	4: //Read back calibration file
		powermoduleCalib.b_StartCalibration := FALSE;
		pulseTimer(IN := NOT JsonFileToStruct(
			bExecute := pulseTimer.Q,
			sJsonPathName := 'C:\PLCUtility\CalDat_Powerstack.json',
			sStructName := 'ST_Powerstack_Calibration',
			pStruct := ADR(st_calibration.Powerstack),
			nStruct := SIZEOF(st_calibration.Powerstack),
			WriteMode := FALSE,
			sMessage => Message,
			Error => bError,
			Busy => bBusy
			));
		IF NOT pulseTimer.IN THEN
			SFCstep := 99;
		END_IF
		
	99: //clear all states for next round
		Error := bError; 
		sMessage := Message;
		pulseTimer.IN := FALSE;
		fbExecuteCalibrationFit(START := FALSE);
		DelayTimer.IN := FALSE;
		fbExecuteCalibrationFit.START := FALSE;
		PowerstackCalibration := TRUE;
		SFCstep := 0;
END_CASE
END_METHOD

METHOD Reset : BOOL
Reset := GenGridControl.Reset();
END_METHOD

METHOD SetPQLimits

VAR_INPUT
	r_BatPchargeLim			: REAL;
	r_BatPdischargeLim		: REAL;
	b_BatteryFull			: BOOL;
	b_BatteryEmpty			: BOOL;
	r_ACLinevoltage			: REAL;
	r_PchargeLimHard		: REAL;
	r_PchargeLimSoft		: REAL;
	r_PDischargeLimHard		: REAL;
	r_PDischargeLimSoft		: REAL;
	r_SmaxHard				: REAL;	//kVA
	r_AmaxHard				: REAL; //current
	r_AmaxSoft				: REAL; //current
END_VAR

VAR_OUTPUT
	r_Pmin				: REAL;
	r_PMax				: REAL;
	r_AMax				: REAL;
END_VAR

VAR_INST
	fb_rampPcharge						: FB_ramp := (b_enable := TRUE, r_ramprate := 25);
	fb_rampPdischarge					: FB_ramp := (b_enable := TRUE, r_ramprate := 25);
	fb_rampCurrentLimit					: FB_ramp := (b_enable := TRUE, r_ramprate := 100);
	
	r_BatChargeCorrectionFactor			: REAL := 0.98; // compensates inverter losses and BMS measurement errors
	r_BatDischargeCorrectionFactor		: REAL := 0.99;
	r_Smax								: REAL;
	r_PDischargeLimitUser				: REAL; //Discharging
	r_PChargeLimitUser					: REAL; //Charging
	r_AmaxLimitUser						: REAL;
	r_PmaxbySmax						: REAL;
	r_BatChargePowerLimitCalc			: REAL;
	r_BatDischargePowerLimitCalc		: REAL;
END_VAR
//user soft limit
fb_rampPcharge(IN := LIMIT(0 ,r_PchargeLimSoft, r_PchargeLimHard));
fb_rampPdischarge(IN := LIMIT(0,r_PDischargeLimSoft, r_PDischargeLimHard));

//current limit
r_AmaxLimitUser := MAX(0, KwToCurrent(r_SmaxHard,r_acLineVoltage), r_AmaxHard);
fb_rampCurrentLimit(IN := LIMIT(0,r_Amaxsoft, r_AmaxLimitUser), Q=> r_AMax);

r_Smax:= CurrentToKw(r_Amax, r_AClinevoltage);
r_PmaxbySmax := r_SMax; //SQRT(MAX(EXPT(r_Smax,2) - EXPT(r_ReaPower, 2),0));

//Set system Variable
r_Pmin := -MIN(ABS(r_BatPchargeLim / r_BatChargeCorrectionFactor), fb_rampPcharge.Q, r_PmaxbySmax);
r_Pmax := MIN(ABS(r_BatPdischargeLim * r_BatDischargeCorrectionFactor),  fb_rampPdischarge.Q, r_PmaxbySmax);

IF b_BatteryFull THEN
	r_Pmin := 0;
ELSIF b_BatteryEmpty THEN
	r_Pmax := 0; //overwrite value from input to 0.
END_IF
END_METHOD

METHOD shutdown : BOOL
VAR_INPUT
END_VAR

VAR_INST
	started : BOOL;
	ton_RetryDelay : TON := (PT := T#2s);
END_VAR
ton_RetryDelay(IN := TRUE);

IF storeSettings(ton_RetryDelay.Q, FALSE) THEN
	shutdown := TRUE;
	ton_RetryDelay(IN := FALSE);
END_IF
END_METHOD

METHOD StoreSettings : BOOL
VAR_INPUT
	execute : BOOL;
	writeMode: BOOL;
END_VAR

VAR_INST
	rTrigExecute	: R_TRIG;
	b_next : BOOL;
	sfcStep	: BYTE;
	tDelaySFCstep		: TON :=(PT := T#10MS);
END_VAR
rTrigExecute(CLK := execute);
IF rTrigExecute.Q THEN
	SFCstep := 1;
END_IF

CASE SFCstep OF
	1: b_next := JsonFileToStruct(
		bExecute := TRUE,
		sJsonPathName := 'C:\PLCUtility\MachineSettings.json',
		sStructName := 'ST_System_MachineParams',
		pStruct := ADR(settings.MachineParams),
		nStruct := SIZEOF(settings.MachineParams),
		WriteMode := writeMode,
		sMessage => sMessage
		);
	2: b_next := JsonFileToStruct(
		bExecute := TRUE,
		sJsonPathName := 'C:\PLCUtility\MachineConfig.json',
		sStructName := 'ST_System_Config',
		pStruct := ADR(settings.Configuration),
		nStruct := SIZEOF(settings.Configuration),
		WriteMode := writeMode,
		sMessage => sMessage
		);
	 3: b_next := JsonFileToStruct(
		bExecute := TRUE,
		sJsonPathName := 'C:\PLCUtility\GridSettings.json',
		sStructName := 'ST_System_GridCodeParams',
		pStruct := ADR(settings.GridParams),
		nStruct := SIZEOF(settings.GridParams),
		WriteMode := writeMode,
		sMessage => sMessage
		);
	 4: b_next := JsonFileToStruct(
		bExecute := TRUE,
		sJsonPathName := 'C:\PLCUtility\MachineProperties.json',
		sStructName := 'ST_System_Properties',
		pStruct := ADR(settings.Properties),
		nStruct := SIZEOF(settings.Properties),
		WriteMode := writeMode,
		sMessage => sMessage
		);
	5: b_next := JsonFileToStruct(
		bExecute := TRUE,
		sJsonPathName := 'C:\PLCUtility\CalDat_Powerstack.json',
		sStructName := 'ST_System_Calibration',
		pStruct := ADR(settings.Calibration),
		nStruct := SIZEOF(settings.Calibration),
		WriteMode := FALSE,
		sMessage => sMessage
		);
	ELSE
		SFCstep := 0;
		rTrigExecute(CLK := FALSE);
		StoreSettings := TRUE;	
END_CASE


IF b_next THEN 
	tDelaySFCstep(IN := TRUE);
 	IF tDelaySFCstep.q THEN 
	SFCstep := SFCstep + 1;
		tDelaySFCstep(IN := FALSE);
	END_IF 
END_IF
END_METHOD

METHOD UpdateSystemTime : BOOL
VAR_INST
	SetTime :	NT_SetLocalTime();
	rtrig_AutoUpdate	:	r_Trig;
	ftrig_UpdateDone	:	f_Trig;
	systime				:	Timestruct;

	SystemTimeStamp		:	DINT;
	GPSTimeStamp		:	DINT;
	TON_GpsUpdateReq	:	TON := (PT := T#5M); 
	
	NewTimeString		:	STRING;
	NewTimeStruct		:	Timestruct;

	
	UpdateRequired		:	BOOL;
END_VAR

monitor.system.DT_SystemTime := GVL.dt_SystemDateTime;

//first fix datetime format from teltonika.
IF st_params.SystemTime.AutoSyncToGPS THEN 
	TON_GpsUpdateReq(in := ABS(DT_TO_DINT(monitor.router.GPS.DateTime) - DT_TO_DINT(gvl.dt_SystemDateTime)) > 30);
	IF ton_gpsUpdateReq.Q THEN
		NewTimeStruct := DT_TO_Systemtime(monitor.Router.GPS.DateTime);
		UpdateRequired	:=	TRUE;
	ELSE
		UpdateRequired	:=	FALSE;
	END_IF
ELSE
	IF st_params.SystemTime.ManualSync THEN
		st_params.SystemTime.ManualSync := FALSE;
		NewTimeStruct := DT_TO_SYSTEMTIME(st_params.SystemTime.ManSyncValue);
		UpdateRequired	:=	TRUE;
	END_IF
END_IF
	
SetTime(	TimeSTR := NewTimeStruct, //convert to Systemtime struct and write to plc
	start	:= UpdateRequired,
	TMOUT	:= T#1S);

			
ftrig_UpdateDone(clk := SetTime.BUSY);

IF ftrig_UpdateDone.Q THEN
	UpdateRequired := FALSE;
	monitor.system.events.b_TimeUpdateFailed := FALSE;
	IF SetTime.ERR THEN
		monitor.system.events.b_TimeUpdateFailed := TRUE;
	END_IF
END_IF
END_METHOD

END_FUNCTION_BLOCK

// ---- POUs/System/PowerControl/FB_PowerControl.TcPOU
FUNCTION_BLOCK FB_PowerControl
VAR_IN_OUT CONSTANT						
	powerstack							: ST_Powerstack_get;
	powermonitor						: ST_powermonitor_get;
	st_params							: ST_Powercontrol_Params;
END_VAR

VAR_INPUT
	r_Soc								: REAL;
	r_SocMin							: REAL;
	r_SocMax							: REAL;
	b_calibrationRun					: BOOL;
	
	
	//inverter data	
	Target								: ST_PowerControl_Target; //input from gengrid controller
	
	r_Pset								: REAL;
	r_Qset								: REAL;
	r_PFset								: REAL;
	b_PFsetEnable						: BOOL;	
	r_Frequency							: REAL;
	r_FreqDroop							: REAL;
	r_Voltage							: REAL;
	r_VoltDroop							: REAL;
	b_GensetLoadshareControl			: BOOL;
	r_GenfixPowerTarget					: REAL;
	r_GenRatedPower						: REAL;
	b_GenStarted						: BOOL;
END_VAR

VAR_OUTPUT
	r_ActivePowerRQInv			: REAL; // Positive discharging, negative charging
	r_ReactivePowerRQInv		: REAL; // Positive  Inductive, negative Capacitive
	r_ActivePowerRQGen			: REAL;
	r_ReactivePowerRQGen		: REAL;
	b_ExtSyncingActive			: BOOL;
	r_FrequencyRQ				: REAL;
	r_VoltageRQ					: REAL;
	r_FreqDroopRQ				: REAL;
	r_VoltDroopRQ				: REAL;
END_VAR
VAR_OUTPUT
	get							: ST_PowerControl_Get;
END_VAR
VAR	
	//General
	VoltageOK				: fbValueOutOfRange;
	ActiveOK				: fbValueOutOfRange;
	ReactiveOK				: fbValueOutOfRange;
	
	//Controlvars
	r_ManSyncPower			: REAL;
	b_Sync					: BOOL;
	r_ReactiveSetpoint		: REAL := 0;
	b_ReactivePIDLimitReached : BOOL;
	
	GensetPeakshaverEnable 	: BOOL;
	r_ActiveSetpoint		: REAL := 0;
	b_ActivePIDLimitReached : BOOL;
	e_ctrl					: e_CTRL_MODE;
	
	b_ReactiveLimit			: BOOL;
	b_ActiveLimit			: BOOL;
END_VAR

//get measured data from peakshaver target or bess netto output.
TargetSection();

//Determine Reactive power setpoint
r_ReactiveSetpoint := PFtoReactiveSetpoint(
	enable := b_PFsetEnable,
	forcezeroQ:= target.b_GenIsoPID,
	voltage := powerstack.r_ACVoltageD7,
	AcCurrentLimit := MAX(target.r_FeedInCurrentLimit, target.r_SupplyCurrentLimit),
	Sact:= get.r_Sact, 
	Qset:= r_Qset,
	PFset:= r_PFset);

//Use droop controller if inverter is in droop mode.
//IF powerstack.e_InverterMode <> eInverterModes.AFE AND powerstack.Netcontactor.b_NetConFb THEN
	DroopController(
		r_NomVolt	:= r_Voltage,
		r_NomFreq	:= r_Frequency,
		r_FreqDroop	:= r_FreqDroop,
		r_VoltDroop	:= r_VoltDroop,
		b_EnableSocDrooping		:= Target.b_EnableSocDrooping AND st_params.SocDroop.enable AND powerstack.b_StartedState,
		r_FreqRQ 		=> r_FrequencyRQ, 
		r_voltRQ 		=> r_VoltageRQ,
		r_FreqDroopRQ	=> r_FreqDroopRQ,
		r_VoltDroopRQ 	=> r_VoltDroopRQ
);
//for letting now powermodule.
b_ExtSyncingActive := target.Syncdata.b_Sync;

//Peakshave power PID controller
IF b_calibrationRun THEN
	Target.PIDmode := ePIDMode.None;
END_IF
PeakshaveController(VoltageOK.Q, ActiveOK.Q, ReactiveOK.Q, Target.PIDmode <> ePIDmode.None AND st_params.ActivePID.enable);

PIDcontrollers(
	b_Activate :=  powerstack.b_ControlEnabled AND powerstack.b_startedstate,
	b_QEnable := (Target.PIDmode = ePIDmode.Q OR Target.PIDmode = ePIDmode.Both) AND st_params.ReactivePID.enable,
	b_PEnable := (Target.PIDmode = ePIDmode.P OR Target.PIDmode = ePIDmode.Both) AND st_params.ActivePID.enable,
	);
	
GensetController(
	Enable := b_GensetLoadshareControl AND b_genstarted,
	GenRatedPower := r_GenRatedPower,
	PeakshaveMode := target.PeakshaveMode,
	ActiveControlEnable := b_activePIDLimitReached OR NOT powerstack.b_startedstate,
	ReactiveControlEnable := b_ReactivePIDLimitReached OR NOT powerstack.b_startedstate,
	Ptarget := -CurrentTokW(target.r_SupplyCurrentLimit, powermonitor.OutputField.ar_LineVoltage[0]),
	PAct := target.Measurements.r_ActivePower,
	PManSet := r_GenfixPowerTarget,
	Qtarget	:= -target.Measurements.r_ReactivePower,
	QactPID := r_ReactivePowerRQInv,
	Pset => r_ActivePowerRQGen,
	Qset => r_ReactivePowerRQGen);
	
//set throttling info	 
ThrottlingInfoSection();

METHOD PRIVATE DroopController : BOOL
VAR_INPUT
	r_NomVolt			: REAL;
	r_NomFreq			: REAL;
	r_FreqDroop			: REAL;
	r_VoltDroop			: REAL;
	b_EnableSocDrooping	: BOOL;
END_VAR

VAR_OUTPUT
	r_FreqRQ				: REAL;
	r_VoltRQ				: REAL;
	r_FreqDroopRQ			: REAL;
	r_VoltDroopRQ			: REAL;
END_VAR

VAR_INST
	b_master				: BOOL := TRUE;
	r_SoCMiddlepoint		: REAL;
	r_FreqZeroCharge		: REAL;
	r_FreqZeroDischarge		: REAL;
	r_SocStartFreqShiftDown : REAL;
	r_SocStartFreqShiftUp   : REAL;

	
	DroopRamp				: fb_ramp := (b_enable := TRUE);
	FreqRamp				: fb_ramp := (b_enable := TRUE);
	VoltRamp				: fb_ramp := (b_enable := TRUE);
	
	
	//freq shift PID
	r_DroopFreqMax			: REAL;
	FreqShiftPID			: fb_ctrl_pid_ext := (eMode := e_Ctrl_mode.eCTRL_MODE_ACTIVE);
	FreqShiftPID_params 	: ST_CTRL_PID_EXT_PARAMS := (
							tCtrlCycleTime := T#10MS,
							tTaskCycleTime := T#2MS);
	r_FreqShiftOut			: REAL;
	
	//Volt shift PID
	r_VoltMaxShiftDelta		: REAL := 40;		
	VoltShiftPID			: fb_ctrl_pid_ext := (eMode := e_Ctrl_mode.eCTRL_MODE_ACTIVE);
	VoltShiftPID_params 	: ST_CTRL_PID_EXT_PARAMS := (
							tCtrlCycleTime := T#10MS,
							tTaskCycleTime := T#2MS);
	r_VoltShiftOut			: REAL;
		
	
END_VAR
r_DroopFreqMax :=  MAX(0.01, powerstack.r_FrequencyDroop) / 100 * settings.GridParams.r_GridNominalFrequency;

r_FreqZeroCharge := r_NomFreq - r_DroopFreqMax;
r_FreqZeroDischarge := r_NomFreq + r_DroopFreqMax;
r_SocStartFreqShiftDown := MAX(r_SocMin, st_params.SocDroop.SocMinDroopStart);
r_SocStartFreqShiftUp   := MIN(r_SocMax, st_params.SocDroop.SocMaxDroopStart);

FreqRamp(r_rampRate := 0.5, SetToIN:= FreqRamp.Q < settings.GridParams.r_GridFrequencyMin);
VoltRamp(r_rampRate := 1, SetToIN := VoltRamp.Q < settings.GridParams.r_GridVoltageMin);
//Voltage set
VoltRamp.IN := LIMIT(settings.GridParams.r_GridVoltageMin, r_Nomvolt, settings.GridParams.r_GridVoltageMax);

//freq shift pid
	VoltShiftPID_params.fkp := st_params.FreqShiftPID.Kp;
	VoltShiftPID_params.tTd := TO_TIME(st_params.FreqShiftPID.Td);
	VoltShiftPID_params.tTn := TO_TIME(st_params.FreqShiftPID.Tn);
	VoltShiftPID_params.tTv := TO_TIME(st_params.FreqShiftPID.Tv);
	VoltShiftPID_params.fOuterWindow := st_params.FreqShiftPID.Outerwindow;
	VoltShiftPID_params.fInnerWindow := st_params.FreqShiftPID.Innerwindow;
	VoltShiftPID_params.fDeadBandOutput := st_params.FreqShiftPID.OutputDeadband;
	VoltShiftPID_params.fDeadBandInput := st_params.FreqShiftPID.InputDeadband;
	VoltShiftPID_params.fOutMaxLimit := r_VoltMaxShiftDelta;
	VoltShiftPID_params.fOutMinLimit := -r_VoltMaxShiftDelta;
	VoltShiftPID(
		fsetPointValue := 0,
		fActualValue := SEL(b_master, powerstack.r_ReactivePower, powerstack.r_ACVoltageD7 - r_NomVolt),
		(*fManSyncValue := powerstack.r_FrequencyD7 - r_NomFreq,
		bSync := FALSE,//powerstack.b_StartedState,*)
		stparams := VoltShiftPID_params);
		//activate simultaniously with freqshift pid.
	IF NOT VoltShiftPID.bError AND NOT target.Syncdata.b_Sync AND st_params.FreqShiftPID.enable AND powerstack.b_StartedState AND powerstack.b_InverterGridFormingMode THEN
		VoltShiftPID.eMode := e_Ctrl_Mode.eCTRL_MODE_ACTIVE;
		r_VoltShiftOut := VoltShiftPID.fOut;
	ELSE
		r_VoltShiftOut := 0;
		VoltShiftPID.eMode := e_Ctrl_Mode.eCTRL_MODE_RESET;
	END_IF
			
//linearly scale frequency down when within soc charge prio and soc min
IF r_soc < r_SocStartFreqShiftDown AND b_EnableSocDrooping THEN
	//Frequency set
	FreqRamp.IN := scale(
		r_in:=r_soc,
		 In_min:= r_SocMin,
		 In_max:= r_SocStartFreqShiftDown,
		 Out_min:= r_FreqZeroCharge,
		 Out_max:= r_NomFreq);
ELSIF r_Soc > r_SocStartFreqShiftUp AND b_EnableSocDrooping THEN
	//Frequency set
	FreqRamp.IN := scale(
		r_in:=r_soc,
		 In_min:= r_SocStartFreqShiftUp,
		 In_max:= r_Socmax,
		 Out_min:= r_NomFreq,
		 Out_max:= r_FreqZeroDischarge);
ELSE
	//Frequency set
	FreqRamp.IN := r_NomFreq;
END_IF

//r_SocFreqShift := FreqRamp.Q - r_NomFreq;

//freq shift pid
	FreqShiftPID_params.fkp := st_params.FreqShiftPID.Kp;
	FreqShiftPID_params.tTd := TO_TIME(st_params.FreqShiftPID.Td);
	FreqShiftPID_params.tTn := TO_TIME(st_params.FreqShiftPID.Tn);
	FreqShiftPID_params.tTv := TO_TIME(st_params.FreqShiftPID.Tv);
	FreqShiftPID_params.fOuterWindow := st_params.FreqShiftPID.Outerwindow;
	FreqShiftPID_params.fInnerWindow := st_params.FreqShiftPID.Innerwindow;
	FreqShiftPID_params.fDeadBandOutput := st_params.FreqShiftPID.OutputDeadband;
	FreqShiftPID_params.fDeadBandInput := st_params.FreqShiftPID.InputDeadband;
	FreqShiftPID_params.fOutMaxLimit := r_DroopFreqMax;
	FreqShiftPID_params.fOutMinLimit := -r_DroopFreqMax;
	FreqShiftPID(
		fsetPointValue := 0,
		fActualValue := powerstack.r_FrequencyD7 - r_NomFreq,
		(*fManSyncValue := powerstack.r_FrequencyD7 - r_NomFreq,
		bSync := FALSE,//powerstack.b_StartedState,*)
		stparams := FreqShiftPID_params);
			
IF NOT FreqShiftPID.bError AND st_params.FreqShiftPID.enable AND powerstack.b_StartedState AND powerstack.e_InverterMode = eInvertermodes.Microgrid THEN
	FreqShiftPID.eMode := e_Ctrl_Mode.eCTRL_MODE_ACTIVE;
	r_FreqShiftOut := FreqShiftPID.fOut;
ELSE
	r_FreqShiftOut := 0;
	FreqShiftPID.eMode := e_Ctrl_Mode.eCTRL_MODE_RESET;
END_IF

r_FreqRQ := LIMIT(r_FreqZerocharge, FreqRamp.Q + r_FreqShiftOut, r_FreqZerodisCharge);
r_VoltRQ := VoltRamp.Q + r_VoltshiftOut;

//overwrite if sync is called
DroopRamp(r_Ramprate := 0.5);
IF target.Syncdata.b_Sync THEN
	DroopRamp.IN :=0.5;
	r_FreqDroopRQ:= DroopRamp.Q;
	r_VoltDroopRQ:= DroopRamp.Q;
	r_freqRQ := target.Syncdata.r_freqSet;
	r_voltRQ := target.Syncdata.r_VoltSet;
ELSE
	DroopRamp.IN := r_FreqDroop;
	r_FreqDroopRQ := MAX(Target.r_droopMinimum,r_FreqDroop);
	r_VoltDroopRQ := MAX(Target.r_droopMinimum, r_VoltDroop);
END_IF
END_METHOD

METHOD EMstop : BOOL
VAR_INPUT
END_VAR
e_ctrl := e_CTRL_MODE.eCTRL_MODE_RESET;
r_ActivePowerRQInv := 0;
r_ReactivePowerRQInv := 0;
END_METHOD

METHOD GensetController : BOOL
VAR_INPUT
	Enable					: BOOL;
	GenRatedPower			: REAL; //kVA
	PeakshaveMode			: BOOL;
	ActiveControlEnable		: BOOL;
	ReactiveControlEnable 	: BOOL;
	PTarget					: REAL;
	PAct					: REAL;
	PManSet					: REAL;
	QTarget					: REAL;
	QActPID					: REAL;
END_VAR

VAR_INST
	//Active powercontrol
	PStepSize 				: REAL := 0.001; //kW
	PDelta					: REAL;
	Pcum					: REAL;
	PlimitReached			: BOOL;
	
	//Reactive powercontrol
	QStepSize 				: REAL := 0.001; //kvar
	QDelta					: REAL;
	Qcum					: REAL;
	

	PFmin					: REAL := 0.8;
	QLimit					: REAL;
	
	GenLimit				: REAL := 90; //%
END_VAR

VAR_OUTPUT
	Pset			: REAL; //in %
	Qset			: REAL; //in %
END_VAR
IF enable THEN
	
	IF ActiveControlEnable AND PeakshaveMode THEN
		PDelta := PTarget - PAct;
		Pcum := LIMIT(0, Pcum + LIMIT(-1, PDelta, 1)* PStepSize, GenLimit);
	ELSE
		Pcum := LIMIT(0, PManSet, ABS(powerstack.r_Pmin));
	END_IF
	
	 
	Qlimit := ABS(Pcum)* ACOS(PFmin);
	
	IF ReactiveControlEnable AND PeakshaveMode THEN
		QDelta := QTarget - QActPID;
		Qcum := LIMIT(-Qlimit, Qcum + QDelta* QStepSize, Qlimit);
	ELSE
		Qcum := 0;
	END_IF
ELSE
	Pcum:= 0;
	Qcum:= 0;
END_IF

Pset := LIMIT(0, Pcum / MAX(1, GenRatedPower) * 100, GenLimit);// percentage limit to 90% of gen power
Qset :=LIMIT(0, Qcum / MAX(1, GenRatedPower) * 100, GenLimit);
END_METHOD

METHOD GetDiagnostics : BOOL
VAR_IN_OUT
	AddError		: ARRAY [*] OF FB_AddErrorST;
	a_ActiveEvents	: ARRAY [*] OF ST_ErrorStruct;
	w_Index			: WORD;
END_VAR
(*Reactive PID error*) 	AddError[w_Index](
		b_ErrorTrig			:= Get.Events.b_ReactivePIDError,
		out_ST_Error			:= a_ActiveEvents[w_Index],
		w_ErrorID				:= 1,
		e_ObjectID				:= eObject_ID.PowerController,
		s_Message				:= 'Reactive PID controller fault.',
		e_sev					:= eseverity.Warning
		);
	w_Index := w_Index +1;
	
(*Active PID error*) 	AddError[w_Index](
		b_ErrorTrig			:= Get.Events.b_ActivePIDError,
		out_ST_Error			:= a_ActiveEvents[w_Index],
		w_ErrorID				:= 2,
		e_ObjectID				:= eObject_ID.PowerController,
		s_Message				:= 'Active PID controller fault.',
		e_sev					:= eseverity.Warning
		);
	w_Index := w_Index +1;
	
(*FreqShift PID error*) 	AddError[w_Index](
		b_ErrorTrig				:= Get.Events.b_ActivePIDError,
		out_ST_Error			:= a_ActiveEvents[w_Index],
		w_ErrorID				:= 3,
		e_ObjectID				:= eObject_ID.PowerController,
		s_Message				:= 'Frequency Shift PID controller fault.',
		e_sev					:= eseverity.Warning
		);
	w_Index := w_Index +1;
END_METHOD

METHOD PRIVATE PeakshaveController : BOOL
VAR_INPUT
	Voltage_OK		: BOOL;
	P_OK			: BOOL;
	Q_OK			: BOOL;
	Enable			: BOOL;
END_VAR

VAR_INST
	FeedLimitCorrection : REAL;
	SupplyLimitCorrection : REAL;
	
	ton_ResetZeroPower : TON := (PT := T#5S);
	r_AppPowerLimIntoSystem		: REAL;
	r_AppPowerLimOutOfSystem	: REAL;
	r_ActivePowerLimIntoSystem	: REAL;
	r_ActivePowerLimOutOfSystem	: REAL;	
	r_PowerDemand				: REAL;
	PIDOK						: BOOL;
	
	r_rampRate					: REAL;
	fbPlimIntoSysRamp			: FB_RAMP := (b_enable := TRUE, r_rampRate := 5); //kw per second)
	fbPlimOutOfSysRamp			: FB_RAMP := (b_enable := TRUE, r_rampRate := 5); //kw per second)
	
END_VAR
//Set slow ramp for genset
r_rampRate:= LIMIT(1, target.r_PIDRampRate, 100);
fbPlimIntoSysRamp(SetZero := NOT (powerstack.b_ControlEnabled AND PIDOK),  r_ramprate := r_rampRate, Q => r_ActivePowerLimIntoSystem,);
fbPlimOutOfSysRamp(SetZero := NOT (powerstack.b_ControlEnabled AND PIDOK), r_ramprate :=  r_rampRate, Q => r_ActivePowerLimOutOfSystem);
ton_ResetZeroPower();
ton_ResetZeroPower.IN := FALSE;

PIDOK := VoltageOK.Q AND ActiveOK.Q AND ReactiveOK.Q AND Enable;
VoltagePeakshavePID(enable:= PIDOK,
	PIDParams := st_params.VoltagePeakshavePID, 
	FeedinLimitCorrection => FeedLimitCorrection, 
	SupplyLimitCorrection => SupplyLimitCorrection);

//power controller sectio
IF PIDOK THEN
	b_Sync := FALSE;
	
	//get active power limits based on the current values.
	r_AppPowerLimIntoSystem := CurrentTokW(LIMIT(0, Target.r_SupplyCurrentLimit - SupplyLimitCorrection, Target.r_SupplyCurrentLimit), get.r_PhaseVoltageAct * 1.73);
	r_AppPowerLimOutOfSystem := CurrentTokW(LIMIT(0, Target.r_FeedInCurrentLimit + FeedLimitCorrection, Target.r_FeedInCurrentLimit), get.r_PhaseVoltageAct * 1.73);
	
	IF target.b_GenIsoPID THEN
		fbPlimIntoSysRamp.IN := r_AppPowerLimIntoSystem;
		fbPlimOutOfSysRamp.IN := r_AppPowerLimOutOfSystem;
	ELSE
		fbPlimIntoSysRamp.IN:= SQRT(ABS(EXPT(r_AppPowerLimIntoSystem,2) - EXPT(get.r_Qact,2))) * SEL(r_AppPowerLimIntoSystem < 0, 1, -1);
		fbPlimOutOfSysRamp.IN:= SQRT(ABS(EXPT(r_AppPowerLimOutOfSystem,2) - EXPT(get.r_Qact,2))) * SEL(r_AppPowerLimOutOfSystem < 0, 1, -1);
	END_IF
	
	r_PowerDemand	:= get.r_Pact - powerstack.r_ActivePower + Target.r_PowerTarget;
	r_activeSetpoint 	:= LIMIT(-r_ActivePowerLimIntoSystem, r_powerDemand, r_ActivePowerLimOutOfsystem);
	
ELSE //If measurements not OK or peakshave target disabled, set manually values.
	//RESET some values
	r_activeSetpoint := r_Pset;
END_IF
END_METHOD

METHOD PRIVATE PFToReactiveSetpoint : REAL
VAR_INPUT
	enable 			: BOOL;
	ForceZeroQ		: BOOL;
	voltage			: REAL;
	Sact			: REAL;
	Qset			: REAL;
	AcCurrentLimit	: REAL;
	PFset			: REAL;
END_VAR

VAR_INST
	PFlimited 	: REAL;
	ReactiveSetpoint	: REAL;
	ApparentPowerLimit: REAL;
END_VAR
ApparentPowerLimit := CurrentToKw(AcCurrentLimit, voltage);

IF enable THEN
	PFlimited := LIMIT(-1, PFset, 1);
	ReactiveSetpoint := Sact * SQRT(1-EXPT(PFset,2))* SEL(PFset < 0, 1, -1);
ELSE
	ReactiveSetpoint := Qset;
END_IF

IF forcezeroQ THEN
	ReactiveSetpoint := 0;
END_IF

PFToReactiveSetpoint := LIMIT(-ApparentPowerLimit, ReactiveSetpoint, ApparentPowerLimit);
END_METHOD

METHOD PRIVATE PIDcontrollers : BOOL

VAR_INPUT
	b_Activate							: BOOL;
	b_QEnable							: BOOL;
	b_PEnable							: BOOL;
END_VAR

VAR_INST
	tnActive					: UINT;
	tnReactive					: UINT;
	
	//triggers
	tonPIDStartDelay		: TON := (PT := T#2S);
	tofPIDSyncHoldDelay		: Tof ;
	r_TriggerReactivePIDMode: R_Trig;
	r_TriggerActivePIDMode	: R_Trig;
	r_TriggerPIDHmiReset	: R_Trig;
	f_TriggerPIDHmiActivate	: F_TRIG;
	
	//Reactive PID
	TranstionReactivePowerRamp			: fb_ramp;	
	fb_PIDReactiveCurrent				: FB_CTRL_PID_EXT;
	st_Params_Reactive					: ST_CTRL_PID_EXT_PARAMS;
	
	
	//Active PID
	TranstionActivePowerRamp			: fb_ramp;
	TransitionSync						: BOOL;	
	fb_PIDActiveCurrent					: FB_CTRL_PID_EXT;
	st_Params_Active					: ST_CTRL_PID_EXT_PARAMS;
	b_DinFbPath							: BOOL; 
	b_ActiveLimitReached				: BOOL;
END_VAR
//set PID RESET/ACTIVE TRIGGER when inverter is running
tonPIDStartDelay(IN:= b_Activate);
tofPIDSyncHoldDelay(IN := target.Syncdata.b_Sync, PT := TO_TIME(st_params.TransitionTime));
r_TriggerReactivePIDMode(CLK:= tonPIDStartDelay.Q AND b_QEnable AND NOT tofPIDSyncHoldDelay.Q);
r_TriggerActivePIDMode(CLK:= tonPIDStartDelay.Q AND b_PEnable AND NOT tofPIDSyncHoldDelay.Q);

IF target.b_GenIsoPID THEN
	tnActive := MAX(100, st_params.ActivePID.Tn * 5);
	tnReactive := MAX(100, st_params.ReactivePID.Tn * 5);
ELSE
	tnActive := st_params.ActivePID.Tn;
	tnReactive := st_params.ReactivePID.Tn;
END_IF


IF r_TriggerReactivePIDMode.CLK THEN
	fb_PIDReactiveCurrent.eMode := e_CTRL_MODE.eCTRL_MODE_ACTIVE;
END_IF

IF r_TriggerActivePIDMode.CLK THEN
	fb_PIDActiveCurrent.eMode := e_CTRL_MODE.eCTRL_MODE_ACTIVE;
END_IF

//RESETS
IF NOT b_PEnable OR NOT b_Activate OR e_ctrl = e_CTRL_MODE.eCTRL_MODE_Reset THEN
	fb_PIDActiveCurrent.eMode := e_CTRL_MODE.eCTRL_MODE_Reset;
END_IF
IF NOT b_QEnable OR NOT b_Activate OR e_ctrl = e_CTRL_MODE.eCTRL_MODE_Reset THEN
	fb_PIDReactiveCurrent.eMode := e_CTRL_MODE.eCTRL_MODE_Reset;
END_IF

//r_TriggerPIDHmiReset(CLK := st_params.PIDreset);
//IF r_triggerPIDHmiReset.Q THEN
//	fb_PIDActiveCurrent.eMode := e_CTRL_MODE.eCTRL_MODE_Reset;
//	fb_PIDReactiveCurrent.eMode := e_CTRL_MODE.eCTRL_MODE_Reset;
//END_IF

//f_TriggerPIDHmiActivate(CLK:= st_params.PIDreset);
//IF f_triggerPIDHmiActivate.Q THEN
//	fb_PIDActiveCurrent.eMode := e_CTRL_MODE.eCTRL_MODE_Active;
//	fb_PIDReactiveCurrent.eMode := e_CTRL_MODE.eCTRL_MODE_Active;
//END_IF

//fb_QlimitMA(IN := LIMIT(0, powerstack.r_Qmax - ABS(powerstack.r_ReactivePower), powerstack.r_Qmax));

	st_Params_reactive.tCtrlCycleTime 		:= T#1MS;
		st_Params_reactive.tTaskCycleTime 	:= T#1MS;
		st_Params_reactive.fKp				:= st_params.ReactivePID.Kp /100;
		st_Params_reactive.tTn				:= TO_TIME(tnReactive);
		st_Params_reactive.tTv				:= TO_TIME(st_params.ReactivePID.Tv);
		st_Params_reactive.tTd				:= TO_TIME(st_params.ReactivePID.Td);
		st_Params_reactive.fOutMaxLimit		:= powerstack.r_RatedPower;
		st_Params_reactive.fOutMinLimit		:= -powerstack.r_RatedPower;
		st_Params_reactive.fDeadBandInput	:=  st_params.ReactivePID.InputDeadband;
		st_Params_reactive.fDeadBandOutput	:=  st_params.ReactivePID.OutputDeadband; //
		st_Params_reactive.finnerwindow		:=  st_params.ReactivePID.Innerwindow; //
		st_Params_reactive.fOuterWindow		:=  st_params.ReactivePID.Outerwindow;
	
	
	fb_PIDReactiveCurrent(
		fSetpointValue 	:=r_ReactiveSetpoint,
		bError			=> get.events.b_ReactivePIDError,
		fActualValue	:= target.Measurements.r_ReactivePower,
		stParams		:=st_Params_reactive);
	
	b_ReactivePIDLimitReached := fb_PIDReactiveCurrent.bMaxLimitReached OR fb_PIDReactiveCurrent.bMinLimitReached;

		//when active PID is started, the sync value must be hold for a while. 
TranstionReactivePowerRamp(IN := powerstack.r_ReactivePower, b_enable:= TRUE, r_ramprate := st_params.TransitionRamp);
fb_PIDReactiveCurrent.fManSyncValue := TranstionReactivePowerRamp.Q;

IF fb_PIDReactiveCurrent.eMode = e_CTRL_MODE.eCTRL_MODE_ACTIVE AND NOT fb_PIDReactiveCurrent.bError THEN
	fb_PIDReactiveCurrent.bSync := TRUE;
	r_ReactivePowerRQInv := fb_PIDReactiveCurrent.fOut; 
ELSIF tofPIDSyncHoldDelay.Q THEN
	fb_PIDReactiveCurrent.bSync := FALSE;
	r_ReactivePowerRQInv := TranstionReactivePowerRamp.Q;
ELSE	
	fb_PIDReactiveCurrent.bSync := FALSE;
	r_ReactivePowerRQInv := r_ReactiveSetpoint;
END_IF


	//ACTIVE POWER PID
	st_Params_Active.tCtrlCycleTime 		:= T#1MS;
		st_Params_Active.tTaskCycleTime 	:= T#1MS;
		st_Params_Active.fKp				:= st_params.ActivePID.Kp / 100;
		st_Params_Active.tTn				:= TO_TIME(tnActive);
		st_Params_Active.tTv				:= TO_TIME(st_params.ActivePID.Tv);
		st_Params_Active.tTd				:= TO_TIME(st_params.ActivePID.Td);
		st_Params_Active.fOutMaxLimit		:= powerstack.r_Pmax;
		st_Params_Active.fOutMinLimit		:= powerstack.r_Pmin;
		st_params_Active.fDeadBandInput		:= st_params.ActivePID.InputDeadband;
		st_Params_Active.fDeadBandOutput	:= st_params.ActivePID.OutputDeadband; //kW
		st_Params_Active.bDInTheFeedbackPath := b_DinFbPath;
		st_params_ACtive.bPInTheFeedbackPath := FALSE;
		st_Params_Active.finnerwindow		:=  st_params.ActivePID.innerwindow;
		st_Params_Active.fOuterWindow		:=  st_params.ActivePID.Outerwindow;
			

	//Active Power PID
	fb_PIDActiveCurrent(
		 fSetpointValue := r_ActiveSetpoint,
		 fActualValue	:=	target.Measurements.r_ActivePower,
		 fManSyncValue := r_ManSyncPower,
		 bError			=> get.events.b_ActivePIDError,
		 stParams		:=st_Params_Active);

	b_ActivePIDLimitReached := fb_PIDactiveCurrent.bMaxLimitReached OR fb_PIDactiveCurrent.bMinLimitReached;
//when active PID is started, the sync value must be hold for a while. 
TranstionActivePowerRamp(IN := powerstack.r_ActivePower, b_enable:= TRUE, r_ramprate := st_params.TransitionRamp);
r_ManSyncPower := TranstionActivePowerRamp.Q;

IF fb_PIDActiveCurrent.eMode = e_CTRL_MODE.eCTRL_MODE_ACTIVE AND NOT fb_PIDActiveCurrent.bError THEN
	IF transitionsync THEN
		fb_PIDActiveCurrent.bSync := TRUE;
		transitionsync:= FALSE;
	ELSE
		fb_PIDActiveCurrent.bSync := b_sync;
	END_IF
	r_ActivePowerRQInv := fb_PIDActiveCurrent.fOut; 
ELSIF tofPIDSyncHoldDelay.Q THEN
	TransitionSync := TRUE;
	fb_PIDActiveCurrent.bSync := FALSE;
	r_ActivePowerRQInv := TranstionActivePowerRamp.Q;
ELSE	
	r_ActivePowerRQInv := r_Pset;
END_IF

b_ActiveLimit := fb_PIDActiveCurrent.bMaxLimitReached OR fb_PIDActiveCurrent.bMinLimitReached;
b_ReactiveLimit := fb_PIDReactiveCurrent.bMaxLimitReached OR fb_PIDReactiveCurrent.bMinLimitReached;
END_METHOD

METHOD Reset : BOOL
e_ctrl := e_CTRL_MODE.eCTRL_MODE_ACTIVE;
END_METHOD

ACTION TargetSection:
VoltageOK(
	r_var := Target.Measurements.r_PhaseVoltage,
	r_Min := settings.GridParams.r_GridVoltageMin / 1.73,
	r_Max := settings.GridParams.r_GridVoltageMax / 1.73,
	r_WhenError := Target.Measurements.r_PhaseVoltage,
	r_Out => get.r_PhaseVoltageAct);
	
ActiveOK(
	r_var := Target.Measurements.r_ActivePower,
	r_Min := -4000,
	r_Max := 4000,
	r_WhenError := Target.Measurements.r_ActivePower,
	r_Out => get.r_Pact);
	
ReactiveOK(
	r_var := Target.Measurements.r_ReactivePower,
	r_Min := -4000,
	r_Max := 4000,
	r_WhenError := Target.Measurements.r_ReactivePower,
	r_Out => get.r_Qact);

get.r_Sact := SQRT(EXPT(get.r_Pact,2) + EXPT(get.r_Qact,2));
get.r_CurrentAct := SEL(get.r_phaseVoltageAct = 0, get.r_Sact * 1000 / (3* get.r_PhaseVoltageAct), 0);
get.r_FeedInCurrentLimitActual := Target.r_FeedInCurrentLimit;
get.r_SupplyInCurrentLimitActual := Target.r_SupplyCurrentLimit;
END_ACTION

ACTION ThrottlingInfoSection:
get.ui_ThrottlingType.0 := Powerstack.PowermoduleMaster.Events.b_CurrThrottlingActive OR Powerstack.PowermoduleSlave.Events.b_CurrThrottlingActive;
get.ui_ThrottlingType.1 := b_ActiveLimit;
get.ui_ThrottlingType.2 := b_ReactiveLimit;
get.ui_ThrottlingType.14 := Powerstack.PowermoduleMaster.Events.b_TempThrottlingActive OR Powerstack.PowermoduleSlave.Events.b_TempThrottlingActive;
get.b_ThrottlingActive := get.ui_ThrottlingType <> 0;
END_ACTION

METHOD VoltagePeakshavePID : BOOL
VAR_INPUT
	Enable				: BOOL;
	PIDParams					: st_Powercontrol_PIDparams;
END_VAR

VAR_INST
	fb_PIDVoltagePowerFeedInLimit	: FB_CTRL_PID_EXT := (eMode := e_CTRL_mODE.eCTRL_MODE_ACTIVE);
	fb_PIDVoltagePowerSupplyLimit	: FB_CTRL_PID_EXT := (eMode := e_CTRL_mODE.eCTRL_MODE_ACTIVE);
	st_Params_VoltagePowerFeedin	: ST_CTRL_PID_EXT_PARAMS := (tCtrlCycleTime := T#1MS,tTaskCycleTime := T#1MS, fkp := 1, tTn:= T#200MS);
	st_Params_VoltagePowerSupply	: ST_CTRL_PID_EXT_PARAMS := (tCtrlCycleTime := T#1MS,tTaskCycleTime := T#1MS, fkp := 1, tTn:= T#200MS);
END_VAR

VAR_OUTPUT
	FeedInLimitCorrection : REAL;
	SupplyLimitCorrection : REAL;
END_VAR
//Common PID params
st_Params_VoltagePowerFeedin.fKp := st_Params_VoltagePowerSupply.fKp := PIDParams.Kp;
st_Params_VoltagePowerFeedin.tTn := st_Params_VoltagePowerSupply.tTn := TO_TIME(PIDParams.Tn);
st_Params_VoltagePowerFeedin.tTd := st_Params_VoltagePowerSupply.tTd := TO_TIME(PIDParams.Td);
st_Params_VoltagePowerFeedin.tTv := st_Params_VoltagePowerSupply.tTv := TO_TIME(PIDParams.Tv);
st_Params_VoltagePowerFeedin.fInnerWindow := st_Params_VoltagePowerSupply.fInnerWindow := PIDParams.InnerWindow;
st_Params_VoltagePowerFeedin.fOuterWindow := st_Params_VoltagePowerSupply.fOuterWindow := PIDParams.OuterWindow;
st_Params_VoltagePowerFeedin.fDeadBandInput := st_Params_VoltagePowerSupply.fDeadBandInput := PIDParams.InputDeadband;

//Supply specific params
st_Params_VoltagePowerFeedIn.fOutMaxLimit := 0;
st_Params_VoltagePowerFeedIn.fOutMinLimit := -Target.r_SupplyCurrentLimit;

fb_PIDVoltagePowerFeedInLimit(
	fSetpointValue := SEL(fb_PIDVoltagePowerFeedInLimit.fOut <> 0, LIMIT(0, powerstack.r_ACVoltageD7 - settings.GridParams.r_GridNominalVoltage, PIDparams.OutputDeadband), PIDparams.OutputDeadband),
	fActualValue := powerstack.r_ACVoltageD7 - settings.GridParams.r_GridNominalVoltage,
	emode := SEL(PIDParams.enable AND Enable, e_CTRL_MODE.eCTRL_MODE_RESET, e_CTRL_MODE.eCTRL_MODE_ACTIVE),
	STParams := st_Params_VoltagePowerFeedIn); 
 
st_Params_VoltagePowerSupply.fOutMaxLimit := Target.r_FeedInCurrentLimit;
st_Params_VoltagePowerSupply.fOutMinLimit := 0;

fb_PIDVoltagePowerSupplyLimit(
	fSetpointValue := SEL(fb_PIDVoltagePowerSupplyLimit.fOut <> 0, LIMIT(-PIDparams.OutputDeadband, powerstack.r_ACVoltageD7 - settings.GridParams.r_GridNominalVoltage, 0), -PIDparams.OutputDeadband),
	fActualValue := powerstack.r_ACVoltageD7 - settings.GridParams.r_GridNominalVoltage,
	emode := SEL(PIDparams.enable AND Enable, e_CTRL_MODE.eCTRL_MODE_RESET, e_CTRL_MODE.eCTRL_MODE_ACTIVE),
	stParams := st_Params_VoltagePowerSupply);
END_METHOD

END_FUNCTION_BLOCK

// ---- POUs/Functions-FBs-Programs/fbValueOutOfRange.TcPOU
FUNCTION_BLOCK fbValueOutOfRange
VAR_INPUT
	r_Min				:REAL;
	r_Max				:REAL;
	r_WhenError			:REAL;
END_VAR

VAR_IN_OUT
	r_var				:REAL;
END_VAR

VAR_OUTPUT
	Q					:BOOL;
	r_Out				:REAL;	
	b_IsError			:BOOL;
END_VAR

IF r_var >= r_Min AND r_var <= r_Max THEN
	Q := TRUE;
ELSE
	Q := FALSE;
	r_var := r_WhenError;
END_IF

b_IsError := NOT Q;
r_Out := r_var;

END_FUNCTION_BLOCK

// ---- POUs/Functions-FBs-Programs/_acFunctions/CurrentToKw.TcPOU
FUNCTION CurrentToKw : REAL
VAR_INPUT
	Current		: REAL;
	linevoltage	: REAL;
END_VAR

IF linevoltage > 100 THEN
	CurrentToKw := (Current * linevoltage * 1.73) / 1000;
ELSE
	CurrentToKw := (Current * 400 * 1.73) / 1000;
END_IF

END_FUNCTION

// ---- POUs/Functions-FBs-Programs/fb_Ramp.TcPOU
FUNCTION_BLOCK fb_Ramp
VAR_INPUT
	SetZero		: BOOL;
	SetToIN		: BOOL;
	IN			: REAL;
	r_ramprate	: REAL;
	b_Enable	: BOOL;
END_VAR
VAR_OUTPUT
	Q		: REAL;
END_VAR

VAR
	r_RampFinal				: REAL;
	fb_ramp					: FB_CTRL_RAMP_GENERATOR;
	st_ParamsRamp    		: ST_CTRL_RAMP_GENERATOR_PARAMS;
	r_inLast				: REAL;
END_VAR

IF SetZero THEN
	IN := 0;
END_IF

IF SETtoIN OR SetZero THEN
	r_RampFinal	:= r_ramprate * 10000;
ELSE
	r_rampFinal := r_ramprate;
END_IF

st_ParamsRamp.fVeloNeg := r_RampFinal;
st_ParamsRamp.fVeloPos := r_RampFinal;
st_ParamsRamp.tCtrlCycleTime := T#1MS;
st_ParamsRamp.tTaskCycleTime := T#1MS;
fb_ramp(
	bEnable:= b_enable,
	fout => Q,
	stParams := st_ParamsRamp,
	fStart:= r_inlast,
	fTarget:= IN);
	

IF fb_ramp.bValueReached AND b_enable THEN
	r_inlast := IN;
END_IF

IF NOT b_enable THEN
	Q := IN;
END_IF

END_FUNCTION_BLOCK

// ---- POUs/System/GenGridControl/FB_GenGridController.TcPOU
FUNCTION_BLOCK FB_GenGridController
VAR_IN_OUT CONSTANT
	monitor						: ST_System_Monitor;
	st_params					: ST_GenGridController_params;
	control						: ST_System_Control;
END_VAR

VAR_INPUT
	Enable						: BOOL;
	b_ForceOperate				: BOOL;
	b_EMSTOP					: BOOL;
END_VAR

VAR_OUTPUT
	TargetData					: ST_PowerControl_Target;
	InverterMode				: eInverterModes;
	PowerMode					: ePowermodes;
	b_inputContactorClose		: BOOL;
	b_inputContactorOpen		: BOOL;
	b_InputSyncEnable			: BOOL;
	b_ExtContactorClose			: BOOL;
	b_IOStartStop				: BOOL;
	b_NetcontactorHoldClose		: BOOL;
	b_ExtGridConnected			: BOOL;
	b_slowLom					: BOOL;
	get							: ST_GenGridController_get;
END_VAR

VAR
	InputContactor				: FB_ContactorControl;
	ExtContactor				: FB_ContactorControl;
	LoadStart					: FB_StartStop := (GreaterThan := TRUE);
	SocStart					: FB_StartStop := (GreaterThan := FALSE);
	ChargeLoadStart				: FB_StartStop := (GreaterThan := TRUE);
	BatFullStart				: FB_StartStop := (GreaterThan := TRUE);	
		
	b_BreakerACok				: BOOL;
	b_BreakerCMDfb				: BOOL;
	b_Breakerfb 				: BOOL;
	ar_BreakerCurrent			: ARRAY[0..4] OF REAL;
	b_InputACOK					: BOOL;
	b_InputMCCBfb				: BOOL;
	b_BusbarACOK				: BOOL;
	b_ExtACOK					: BOOL;
	b_SFCmodetransInhibit		: BOOL;
	b_GridCodeTripInverter		: BOOL;
	b_GridCodeActive			: BOOL;
	b_GridACDetected			: BOOL;
	b_SkipGensetCooldown		: BOOL;
	b_loadbankEnable			: BOOL;
	b_hybridMode				: BOOL;
	b_ManGenStartStop			: BOOL;
	b_GridTakeOverMode			: BOOL;
	b_AMFEnabled				: BOOL;
	b_autoSwitching				: BOOL;
	b_GenStarted				: BOOL;
	b_GenfreqProtection			: BOOL;
	GenFailCounter				: CTU;
	b_GridcodeOK				: BOOL;
	b_AFEActive					: BOOL;
	r_Soc						: REAL;
	r_ACVoltageBusbar			: REAL;
	b_PSBActive					: BOOL;	
	b_BESSReady					: BOOL;		
	 
	//Scheduler
	b_TimeSlot1					: BOOL;
	b_TimeSlot2					: BOOL;
	
	//Signals
	SFCEnable					: BOOL := TRUE;
	b_StartCondition			: BOOL;
	SFCTransTrigger			: TON := (PT :=T#10MS);
	SFCResetTrigger				: BOOL; // from inside SFC itself
	
	//Genset
	GensetSetpoints				: ST_Genset_Setpoints;
	t_CooldownTime				: TIME;
	t_WarmupTime				: TIME;
	
	//ControlModes
	b_ActivateTransition		: BOOL;
	b_ActivatePowerControl		: BOOL;
	eModeLocal 					: (AFE, UgridDroop, UgridIso, UgridIsland);
	PowerControlMode			: ePowerControlmode;
	BreakerOperationMode		: eBreakerOperationMode;
	ExtGensetEnable				: BOOL;
	
	// future work : eGenPowerTarget 				: (minimum, efficiency, maximum);
END_VAR

//FIRST SETUP IO
InputContactor(monitor := monitor, control := control, SyncData := targetdata.Syncdata, st_params := st_params.Contactor,
	b_FbIn := monitor.ACswitchgear.b_InputContactorfb,
	r_AcVoltageRef := monitor.powermonitor.InputField.ar_LineVoltage[0],
	r_AcFreqRef := monitor.powermonitor.InputField.ar_Frequency[0],
	li_VoltCrossRef := monitor.powermonitor.InputField.li_TimeVoltZeroCrossup,
	li_VoltCrossBus := monitor.peakshavebox.Powermonitor.li_TimeVoltZeroCrossup,
	e_AcRotationRef := monitor.powermonitor.InputField.e_ACrotationStatus,
	e_AcRotationBus := monitor.powermonitor.Outputfield.e_ACrotationStatus,
	b_SyncOK := monitor.ACswitchgear.b_InputSynchronizerfb,
	b_deloadEnable := TRUE,
	ar_current := Monitor.powermonitor.InputField.ar_Current,
	r_Power := Monitor.powermonitor.InputField.ar_ActivePower[0],
	CloseCMD => b_inputContactorClose,
	OpenCMD	=> b_inputContactorOpen,
	SyncEnable => b_InputSyncEnable,
	RotationFault => get.events.b_RotationFieldFault,
	b_deadbus := NOT b_BusbarACOK,
);

ExtContactor(monitor := monitor, control := control, syncdata := targetdata.Syncdata, st_params := st_params.Contactor,
	b_FbIn := monitor.peakshavebox.b_ContactorFb,	 
	r_AcVoltageRef:= monitor.peakshavebox.Powermonitor.ar_LineVoltage[0],
	r_AcFreqRef := monitor.peakshavebox.Powermonitor.ar_Frequency[0],
	li_VoltCrossRef := monitor.peakshavebox.Powermonitor.li_TimeVoltZeroCrossup,
	b_SyncOK := monitor.peakshavebox.b_SyncFb,
	b_deloadEnable := FALSE,
	ar_current := Monitor.peakshavebox.Powermonitor.ar_Current,
	CloseCMD => b_ExtContactorClose,
	b_deadbus := NOT b_BusbarACOK
);

//Map monitor vars to local vars for clearity.
b_ExtACOK := ExtContactor.ACok;
b_InputACOK := InputContactor.ACok AND monitor.ACswitchgear.b_InputMCCBfb AND NOT InputContactor.RotationFault;
b_InputMCCBfb := monitor.ACswitchgear.b_InputMCCBfb;
b_BusbarACOK :=  ACcheck(monitor.powerstack.r_ACVoltageD7 , monitor.powerstack.r_FrequencyD7);
r_ACVoltageBusbar := monitor.powerstack.r_ACVoltageD7;
b_AFEActive	:= monitor.powerstack.b_StartedState AND monitor.powerstack.e_InverterMode = einvertermodes.Afe;
b_TimeSlot1 := control.SoftSettings.system.ScheduleTimeSlot1.b_active;
b_TimeSlot2 := control.SoftSettings.system.ScheduleTimeSlot2.b_active;
SFCEnable := BreakerOperationMode <> eBreakerOperationMode.none AND enable AND NOT get.b_faultActive AND NOT b_EMStop;
b_GridCodeTripInverter := NOT monitor.powerstack.b_GridCodeOK;
b_loadbankEnable := control.softSettings.inputgenset.Loadbank.b_Enable;
b_hybridMode := control.softsettings.inputgenset.b_HydridMode;
b_GridTakeOverMode := (control.Operation.system.b_GridTakeOverEnable AND control.SoftSettings.setup.e_AcInputType = eACInputType.Grid);
get.e_GensetStartStop := GensetStartStop(control.softSettings.inputgenset.b_AutoStartStop, control.Operation.Genset.b_manualStart); 
b_AMFEnabled := control.SoftSettings.system.b_AMF;
//b_AutoResyncGridReco := control.SoftSettings.inputgrid.b_AutoResyncAfterGridRecovery;
b_autoSwitching	:= control.SoftSettings.inputgrid.breaker.AutoConnect;
t_CooldownTime := TO_TIME(TO_DINT(control.softSettings.inputgenset.Generator.ui_CooldownTime) * 60000);
t_WarmUpTime := TO_TIME(TO_DINT(control.softSettings.inputgenset.Generator.ui_WarmupTime) * 60000);
b_GenfreqProtection	:= control.SoftSettings.inputgenset.b_FreqProtectionEnable;
r_soc := Monitor.battery.BatteryInfo.r_SOCScaled;
b_GridCodeActive := control.SoftSettings.inputgrid.b_GridCodesActive;//monitor.powerstack.b_GridCodeCheckActive;
b_GridAcDetected := monitor.powerstack.b_GridACdetected;
b_BreakerACok := SEL(BreakerOperationMode = eBreakerOperationMode.ExtGrid, b_InputACOK, b_ExtACOK);
b_BreakerCMDfb := SEL(BreakerOperationMode = eBreakerOperationMode.ExtGrid, b_inputContactorClose, b_ExtContactorClose);
b_Breakerfb := SEL(BreakerOperationMode = eBreakerOperationMode.ExtGrid, inputcontactor.b_fb, extcontactor.b_fb);
ar_BreakerCurrent := SEL(BreakerOperationMode = eBreakerOperationMode.ExtGrid, inputcontactor.ar_current, extcontactor.ar_current);
b_ActivateTransition := control.Operation.system.b_GenGridModeTrans;
b_PSBActive := monitor.peakshavebox.b_active;
b_BESSReady := monitor.powerstack.b_StartedState;
StartStopConditions((SFCenable OR control.softSettings.setup.b_ExtGenset) AND monitor.powerstack.b_ControlEnabled);

GetControlTarget(
	control:= control,
	monitor := monitor,
	PowerControlMode := PowerControlMode,
	TargetData := TargetData,
	GensetSetpoints := GensetSetpoints,
	b_SFCPIDActivation:= b_ActivatePowerControl,
	b_deload := Inputcontactor.b_Deload OR ExtContactor.b_Deload,
	b_PSBactive := b_PSBactive);

SetBreakerAndPowercontrolMode(
	ACInputType := control.SoftSettings.setup.e_AcInputType,
	GridMode:= control.SoftSettings.setup.e_Gridmode,
	GensetMode := control.softSettings.inputgenset.Generator.e_GensetMode,
	PSBMode := monitor.peakshavebox.PSBmode,
	PSBenable := b_PSBActive, // control.SoftSettings.setup.b_PeakshaveBoxEnable,
	b_Extgenset := control.SoftSettings.setup.b_ExtGenset,
	PowerControlMode := PowerControlMode,
	ExtGensetMode := ExtGensetEnable);
	
SetInverterMode(
	Gridmode := control.SoftSettings.setup.e_Gridmode,
	UgridPowerMode := control.SoftSettings.system.e_UgridPowerMode,
	BreakerMode := BreakerOperationMode,
	PSBMode := monitor.peakshavebox.PSBmode,
	b_inputGridCodeEnabled := b_GridCodeActive AND NOT b_GridTakeOverMode,
	b_gridacDetected := b_GridACDetected, 
	b_PowerstackStarted := monitor.powerstack.b_StartedState,
	b_extFb := ExtContactor.b_fb,
	b_InputFb := InputContactor.b_fb,
	b_AMF := b_AMFEnabled)
;

//SFC actions
SFCtransTrigger(); //timer
GenGridSFC();

//ExtGenset control
ExtGensetControl(
	soft := control.SoftSettings.inputgenset,
	setpoints := gensetsetpoints,
	ExtGensetEnable);

//Get events that give fault states and reset SFC
BundleFaultEvents(events := get.events);

//some resets
SFCReset := NOT SFCEnable OR SFCResetTrigger;
IF NOT monitor.powerstack.b_StartedState THEN
	Genfailcounter.RESET := TRUE;
END_IF

METHOD BundleFaultEvents : BOOL
VAR_IN_OUT
	events : ST_GenGridController_Events;
END_VAR
get.b_faultActive := 
	//events.b_OverFreqTrip 				OR
	//events.b_UnderFreqTrip				OR
	events.b_StartupFault				OR
	events.b_SynchronisationFault 		OR
	events.b_WarmupFault;
	//events.b_OverloadTrip;

IF get.b_faultActive THEN
	get.e_state := eGenGridState.Init;
END_IF

IF BreakerOperationMode <> eBreakerOperationmode.GridFeedthrough OR BreakerOperationMode <> eBreakerOperationmode.ExtGrid THEN
	events.b_GridLostTrip := FALSE;
END_IF
END_METHOD

ACTION ContinousActions:
//if AMF is enabled, netcontactor must always stay closed.
IF monitor.powerstack.b_ControlEnabled AND (BreakerOperationMode <> eBreakerOperationMode.None AND BreakerOperationMode <> eBreakerOperationMode.GenFix) THEN
	b_NetcontactorHoldClose := b_AMFEnabled;
ELSE
	b_NetcontactorHoldClose := FALSE;
END_IF
END_ACTION

METHOD Cooldown : BOOL
VAR_INPUT
	SynchroneGenMode	: BOOL;
END_VAR

VAR_INST
	t_time				: TIME;
	b_stopfb			: BOOL;
	ton_StopTimeOut		: TON;
	ton_CoolDownTimeOut	: TON;
	tp_releaseTimer		: Tp := (PT := T#20MS);
	r_CurrentThresholdShutdown: REAL := 10;
	b_CurrentDown		: BOOL;
	b_release			: BOOL;
END_VAR
get.e_state := eGenGridState.Cooldown;
b_release := FALSE;

IF b_SkipGensetCooldown THEN
	ton_StopTimeOut.PT := T#0S;
ELSE
	ton_StopTimeOut.PT :=t_CooldownTime;
END_IF

//Set timers for cooldown and cooldown time out (if nothing happens when stop is given).
ton_StopTimeOut(IN := b_breakerACOK AND b_CurrentDown AND NOT ton_StopTimeOut.Q); 
b_CurrentDown := monitor.powermonitor.InputField.ar_Current[0] < r_CurrentThresholdShutdown;
ton_CoolDownTimeOut(IN:= NOT b_CurrentDown AND NOT b_IOStartStop AND NOT ton_CoolDownTimeOut.Q, PT:=t_CooldownTime + T#3M);

IF SynchroneGenMode THEN
	b_IOStartStop := FALSE;
	get.b_gensetHot := FALSE;
	b_release := NOT b_IOStartStop AND b_CurrentDown OR ton_CoolDownTimeOut.Q;
ELSE
	IF ton_StopTimeOut.Q OR NOT b_breakerACOK THEN
		ton_StopTimeOut.IN := FALSE;
		b_IOStartStop := FALSE;	
		b_release := TRUE;
		get.b_gensetHot := FALSE;
	END_IF
END_IF

IF ton_CoolDownTimeOut.Q THEN
	get.events.b_ShutdownTimeOut := TRUE;	
END_IF

tp_releaseTimer(IN :=b_release AND NOT tp_releaseTimer.Q, Q => COOLDOWN);
//cooldown := b_release;
END_METHOD

METHOD CurrentLimitProtection : BOOL
VAR_INPUT
	enable				: BOOL;
	FeedinLimit 		: REAL;
	SupplyLimit			: REAL;
	Current				: REAL;
	Power				: REAL;
	TripDelay			: TIME := T#5S;
END_VAR

VAR_INST
	Direction			: SINT;
	ton_DelayTimer		: TON;
END_VAR
ton_DelayTimer(PT := TripDelay, Q => CurrentLimitProtection);

IF Current * LIMIT(-1, power, 1) < 0 AND enable THEN
	ton_DelayTimer.IN := ABS(Current) > ABS(supplyLimit + st_params.by_CurrentLimitMargin);
ELSIF Current * LIMIT(-1, power, 1) > 0 AND enable THEN
	ton_DelayTimer.IN := ABS(Current) > ABS(feedinLimit + st_params.by_CurrentLimitMargin);
ELSE
	ton_DelayTimer.IN := FALSE;
END_IF
END_METHOD

METHOD ExtGensetControl : BOOL

VAR_IN_OUT CONSTANT
	soft		: ST_SoftSettings_Genset;
END_VAR

VAR_IN_OUT
	setpoints 	: ST_Genset_setpoints;
END_VAR

VAR_INPUT
	enable				: BOOL;
END_VAR

VAR_INST
	trip				: BOOL;
	rtrigreset			: R_TRIG;
END_VAR
IF enable THEN
	get.e_GensetMode := eGensetmode.FixedPower;
	IF b_TimeSlot2 THEN
		setpoints := soft.setpointTimeslot2;
	ELSE 
		setpoints := soft.setpointTimeslot1;
	END_IF
	
	//set trip
	trip := GenFreqVoltProtections(TRUE, TRUE ,NOT enable OR control.control.b_Reset, 0);
	
	IF trip THEN
		b_IOstartstop := FALSE;
	ELSE
		b_IOstartStop := b_startcondition;
	END_IF	
END_IF
 
	//Reset OCP trip
rTrigReset(CLK := NOT enable OR control.control.b_Reset);
IF rtrigReset.Q THEN
	b_IOstartstop := FALSE;
END_IF
END_METHOD

METHOD ExtIOControl : BOOL
VAR_INPUT
	r_Power	: REAL;
	r_RatedPower : REAL;
END_VAR
END_METHOD

METHOD GenDownCheck : BOOL
VAR_INPUT
	enable				: BOOL;
	reset				: BOOL;
END_VAR

VAR_INST
	GenFailLimitReached			: BOOL;
	r_ActivePower				: REAL;
	ton_FlatZeroPowerTimeOut 	: TON := (PT:= T#3S);
	ton_reversePowerTrip		: TON := (PT:= T#1S);
	ton_EnableRelease			: TON := (PT:= T#2S);
	ton_GenStartTimeOut			: TON := (PT:= T#1M);
	
	rTrigStarted				: R_Trig;
	
	GenDown						: BOOL;
	i_reversePowerThreshold		: INT := 10; 
	r_FreqLowLimit				: REAL := 49;
	
	GendownTrigger				: STRING;
END_VAR
r_ActivePower := monitor.powermonitor.InputField.ar_ActivePower[0];

//rTrigStarted(CLK :=  r_ActivePower > 1 OR r_ActivePower < -1);
IF r_ActivePower > 1 OR r_ActivePower < -1 THEN
	b_genStarted := TRUE;
END_IF

ton_GenStartTimeOut(IN := ton_EnableRelease.Q AND NOT b_genStarted);
IF ton_GenStartTimeOut.Q THEN
	get.events.b_StartupFault := TRUE;
END_IF

IF reset AND NOT get.events.b_GenDownTrip THEN
	GenDown := FALSE;
	GendownTrigger := '';
	ton_FlatZeroPowerTimeOut.IN := FALSE;
	ton_reversePowerTrip.IN := FALSE;
END_IF

ton_EnableRelease(IN := enable);
ton_reversePowerTrip();
ton_FlatZeroPowerTimeOut();

IF ton_EnableRelease.Q THEN
	ton_reversePowerTrip.IN := NOT b_loadbankEnable AND r_ActivePower > i_reversePowerThreshold;
	ton_FlatZeroPowerTimeOut.IN := LIMIT(-0.5, r_ActivePower, 0.5) = r_ActivePower AND NOT RESET AND b_breakerFB AND b_IOStartStop AND b_GenStarted;
ELSE
	ton_reversePowerTrip.IN := FALSE;
	ton_FlatZeroPowerTimeOut.IN := FALSE;
END_IF

IF (*ton_FlatZeroPowerTimeOut.Q*) ZeroCurrentDisconnect() THEN
	GenDownTrigger := 'zero power trigger';
ELSIF ton_reversePowerTrip.Q THEN
	GenDownTrigger := 'reverse power trigger';
ELSIF SEL(b_GenfreqProtection, FALSE, GenFreqVoltProtections(FALSE, GenFailLimitReached, reset, r_ActivePower)) THEN
	GenDownTrigger := 'Frequency protections trigger';
END_IF

IF GenDownTrigger <> '' THEN	
	IF GenFailLimitReached THEN
		get.events.b_GenDownTrip := TRUE;
	END_IF	 
	GenDown := TRUE;
	b_genStarted := FALSE;
END_IF

GenFailCounter(CU := GenDown, PV := st_params.Genset.GenDownRetries, Q=>GenFailLimitReached, RESET := reset AND get.events.b_GenDownTrip);

IF NOT b_IOStartStop THEN
	b_genStarted := FALSE;
END_IF
GenDownCheck := GenDown;
END_METHOD

METHOD GenFreqVoltProtections : BOOL
VAR_INPUT
	FixedPowerOverloadProtect : BOOL;
	enableEvents	: BOOL;
	reset : BOOL;
	Power : REAL;
END_VAR

VAR_INST
	ton_OCPDelay			: TON := (PT := T#3S);
	ton_OverFreqTripDelay 	: TON := (PT := T#3S);
	ton_UnderFreqTripDelay 	: TON := (PT := T#3S);
	ton_OverVoltTripDelay 	: TON := (PT := T#3S);
	ton_UnderVoltTripDelay 	: TON := (PT := T#3S);
	b_TripDetected			: BOOL;
END_VAR
ton_UnderFreqTripDelay(PT := TO_TIME(ST_params.Genset.UnderfrequencyTripDelay));
ton_OverFreqTripDelay(PT := TO_TIME(ST_params.Genset.OverfrequencyTripDelay));
ton_UnderVoltTripDelay(PT := TO_TIME(ST_params.Genset.UnderVoltageTripDelay));
ton_OverVoltTripDelay(PT := TO_TIME(ST_params.Genset.OverVoltageTripDelay));
ton_OCPDelay(PT := TO_TIME(ST_params.Genset.OverloadTripDelay));

IF reset THEN
	ton_OverFreqTripDelay.IN := FALSE;
	ton_UnderFreqTripDelay.IN := FALSE;
	ton_OverVoltTripDelay.IN := FALSE;
	ton_UnderVoltTripDelay.IN := FALSE;
	ton_OCPDelay.IN := FALSE;
ELSIF monitor.powerstack.b_StartedState THEN
	//Overfrequency protection
	ton_OverFreqTripDelay.IN := monitor.powerstack.r_FrequencyD7 > st_params.Genset.OverFrequencyLimit;
	IF ton_OverFreqTripDelay.Q THEN
		get.events.b_OverFreqTrip := TRUE;
	END_IF
	
	ton_UnderFreqTripDelay.IN := monitor.powerstack.r_FrequencyD7 < st_params.Genset.UnderFrequencyLimit;
	IF ton_UnderFreqTripDelay.Q THEN
		get.events.b_UnderFreqTrip := TRUE;
	END_IF
	
	ton_OvervoltTripDelay.IN := monitor.powerstack.r_ACVoltageD7 > st_params.Genset.OverVoltageLimit AND NOT FixedPowerOverloadProtect;
	IF ton_OverVoltTripDelay.Q THEN
		get.events.b_OverVoltTrip := TRUE;
	END_IF
	
	ton_UnderVoltTripDelay.IN := monitor.powerstack.r_ACVoltageD7 < st_params.Genset.UnderVoltageLimit AND NOT FixedPowerOverloadProtect;
	IF ton_UnderVoltTripDelay.Q THEN
		get.events.b_UnderVoltTrip := TRUE;
	END_IF
	
	//Overcurrent protection
	ton_OCPDelay.IN := FixedPowerOverloadProtect AND monitor.powerstack.r_LoadPercent > monitor.powerstack.r_OvercurrentValueAct * 100 AND monitor.powerstack.e_PowerState = ePowerstate.Charging;
	IF ton_OCPDelay.Q THEN
		get.events.b_OverloadTrip := TRUE;
	END_IF
END_IF

b_TripDetected := get.events.b_OverloadTrip 
	OR get.events.b_OverFreqTrip 
	OR get.events.b_UnderFreqTrip
	OR get.events.b_OverVoltTrip
	OR get.events.b_UnderVoltTrip;

IF NOT enableEvents THEN
	get.events.b_OverFreqTrip := FALSE;
	get.events.b_OverloadTrip := FALSE;
	get.events.b_OverVoltTrip := FALSE;
	get.events.b_UnderVoltTrip := FALSE;
	get.events.b_UnderFreqTrip := FALSE;
END_IF

GenFreqVoltProtections := b_TripDetected;
END_METHOD

ACTION GenGridSFC:
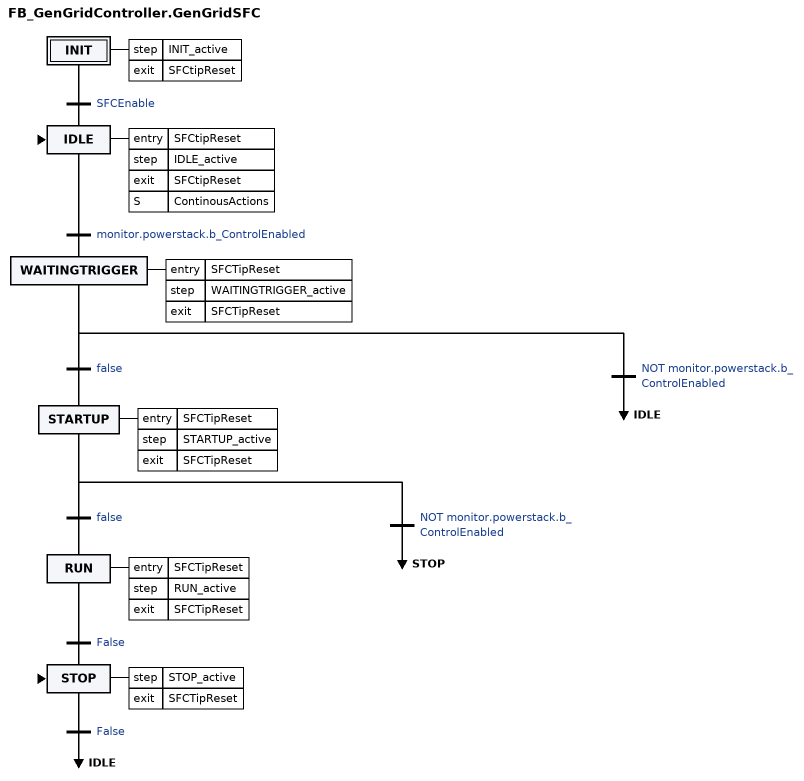
INITIAL_STEP INIT:  // min time T#2s
    INIT_active(N);  // step action
    SFCtipReset(P0);  // exit action
END_STEP
TRANSITION FROM INIT TO IDLE
    := SFCEnable;
END_TRANSITION
STEP IDLE:  // min time T#1s
    SFCtipReset(P1);  // entry action
    IDLE_active(N);  // step action
    SFCtipReset(P0);  // exit action
    ContinousActions(S);
END_STEP
TRANSITION FROM IDLE TO WAITINGTRIGGER
    := monitor.powerstack.b_ControlEnabled;
END_TRANSITION
STEP WAITINGTRIGGER:  // min time T#1s
    SFCTipReset(P1);  // entry action
    WAITINGTRIGGER_active(N);  // step action
    SFCTipReset(P0);  // exit action
END_STEP
TRANSITION FROM WAITINGTRIGGER TO STARTUP
    := false;
END_TRANSITION
TRANSITION FROM WAITINGTRIGGER TO IDLE
    := NOT monitor.powerstack.b_ControlEnabled;
END_TRANSITION
STEP STARTUP:  // min time T#100ms
    SFCTipReset(P1);  // entry action
    STARTUP_active(N);  // step action
    SFCTipReset(P0);  // exit action
END_STEP
TRANSITION FROM STARTUP TO RUN
    := false;
END_TRANSITION
TRANSITION FROM STARTUP TO STOP
    := NOT monitor.powerstack.b_ControlEnabled;
END_TRANSITION
STEP RUN:  // min time T#50ms
    SFCTipReset(P1);  // entry action
    RUN_active(N);  // step action
    SFCTipReset(P0);  // exit action
END_STEP
TRANSITION FROM RUN TO STOP
    := False;
END_TRANSITION
STEP STOP:  // min time T#2s
    STOP_active(N);  // step action
    SFCTipReset(P0);  // exit action
END_STEP
TRANSITION FROM STOP TO IDLE
    := False;
END_TRANSITION
// branch label Branch0_GenGridSFC
// branch label Branch1_GenGridSFC
END_ACTION

METHOD GensetStartStop : eGensetStartStop
VAR_INPUT
	b_autoMode : BOOL;
	b_ManStartStop : BOOL;
END_VAR

VAR_INST
	rTRIG_StartStop	: r_TRIG;
	ManualStart		: BOOL;
	StateInAutoMode	: BOOL;
	GensetTransInhibit: BOOL;
END_VAR
rTRIG_StartStop(CLK := b_ManStartStop);
IF rTRIG_StartStop.Q THEN
	ManualStart := NOT ManualStart;
	StateInAutoMode := FALSE;
END_IF

IF get.e_state = eGenGridState.Idle AND get.b_ModeTransActive THEN
	ManualStart := FALSE;
END_IF


IF b_AutoMode AND NOT get.events.b_TransFromInputGenAckRQ THEN
	GensetStartStop := eGensetStartStop.Auto;
	StateInAutoMode := b_IOstartStop;
ELSE
	IF ManualStart OR StateInAutoMode THEN
		GensetStartStop := eGensetStartStop.Start;
	ELSE
		GensetStartStop := eGensetStartStop.Stop;	
	END_IF
END_IF
END_METHOD

METHOD GetControlTarget

VAR_IN_OUT CONSTANT
	Control					: ST_System_Control;
	monitor					: ST_System_Monitor;
END_VAR

VAR_IN_OUT
	TargetData				: ST_PowerControl_Target;
	GensetSetpoints			: ST_Genset_Setpoints;
END_VAR

VAR_INPUT
	PowerControlMode			: ePowerControlMode;
	b_SFCPIDActivation			: BOOL;
	b_Deload					: BOOL;
	b_PSBactive					: BOOL;
END_VAR

VAR_INST
	b_PSBActiveConditions	: BOOL;
	b_SFCDeactivationEnable : BOOL;
	b_SoCTargetEnable		: BOOL;
	b_inputOvercurrent		: BOOL;	
	r_activePowerMeas		: REAL;
	
	r_MaxActive				: REAL;			
END_VAR
b_PSBActiveConditions := monitor.peakshavebox.b_active AND b_ExtACOK;
b_SFCDeactivationEnable := TRUE;
b_SoCTargetEnable := control.HardSettings.setup.e_ControlSource = eControlsources.Local AND NOT control.Operation.system.b_GridTakeOverEnable;

CASE PowerControlMode OF
	ePowerControlMode.None:
		Targetdata.Measurements.r_ActivePower := monitor.powermonitor.OutputField.ar_ActivePower[0];
		Targetdata.Measurements.r_ReactivePower := monitor.powermonitor.OutputField.ar_ReactivePower[0];
		Targetdata.Measurements.r_PhaseVoltage := 0;
		IF inputcontactor.b_fb OR monitor.powerstack.b_InverterGridFormingMode THEN
			Targetdata.PIDmode := ePIDmode.None;
		ELSE
			Targetdata.r_FeedInCurrentLimit := 1000;
			Targetdata.r_SupplyCurrentLimit := 1000;
			Targetdata.PIDmode := ePIDmode.Both;
		END_IF
		Targetdata.b_GenIsoPID := FALSE;
		Targetdata.r_droopMinimum := 0;
		b_SFCDeactivationEnable := FALSE;	
		
//Grid extern peakshaver
	ePowerControlMode.PeakshaveExt: 
		//peakshave ext genset in droop
		IF control.softsettings.inputgenset.b_PSBExtGensetMonitoring THEN
			TargetData := MapGensetTarget(
				soft := control.SoftSettings.inputgenset,
				r_activePower := monitor.peakshavebox.Powermonitor.ar_ActivePower[0],
				r_reactivePower := monitor.peakshavebox.Powermonitor.ar_ReactivePower[0],
				r_Phasevoltage	:= monitor.peakshavebox.Powermonitor.ar_LineVoltage[0],
				b_active := b_PSBActiveConditions AND monitor.powerstack.b_StartedState AND b_IOstartstop, //IF PSB added, this must be activated by HMI toggle button or something.
				setpoints := Gensetsetpoints);
		ELSE
			IF BreakerOperationMode = eBreakerOperationmode.GridFeedthrough THEN
				//Check inputsection for overcurrent, to be used later
			b_InputOvercurrent := ValueOutOfRange(
				r_min := 0,
				r_max := control.SoftSettings.inputgrid.setpointTimeslot1.r_supplyCurrentLimitSoft,
				r_var := monitor.powermonitor.InputField.ar_Current[0]);
			ELSE
				b_inputOvercurrent := FALSE;
			END_IF
			
			TargetData := MapGridTarget(
				slot1 := control.SoftSettings.PSB.setpointTimeslot1,
				slot2 := control.SoftSettings.PSB.setpointTimeslot2,
				r_activePower := monitor.peakshavebox.Powermonitor.ar_ActivePower,
				r_reactivePower := monitor.peakshavebox.Powermonitor.ar_ReactivePower,
				r_Phasevoltage	:= monitor.peakshavebox.Powermonitor.ar_PhaseVoltage[0],
				Peakshavemode := control.SoftSettings.PSB.PeakshaveMode,
				r_feedInCurrentLimit:= monitor.peakshavebox.r_MaxCTCurrent,
				r_supplyCurrentLimit:= monitor.peakshavebox.r_MaxCTCurrent,
				b_active := b_PSBActiveConditions AND SEL(control.SoftSettings.psb.b_BreakerControl,TRUE, monitor.peakshavebox.b_ContactorFb)
					AND NOT monitor.powerstack.b_InverterGridFormingMode
					AND monitor.powerstack.b_StartedState,
				b_enableSocTarget := b_SoCTargetEnable);
				b_SFCDeactivationEnable := control.softsettings.psb.b_BreakerControl;
		END_IF
	


//Grid input peakshaver
	ePowerControlMode.PeakshaveInputGrid:
		r_MaxActive := MIN(monitor.powermonitor.InputField.ar_ActivePower[1], monitor.powermonitor.InputField.ar_ActivePower[2], monitor.powermonitor.InputField.ar_ActivePower[3]) * 3;		
		
		TargetData := MapGridTarget(
			slot1 := control.SoftSettings.inputgrid.setpointTimeslot1,
			slot2 := control.SoftSettings.inputgrid.setpointTimeslot2,
			r_activePower := monitor.powermonitor.InputField.ar_ActivePower,						
			r_reactivePower := monitor.powermonitor.InputField.ar_ReactivePower,
			r_Phasevoltage	:= monitor.powermonitor.InputField.ar_PhaseVoltage[0],
			Peakshavemode := control.SoftSettings.inputgrid.PeakshaveMode,
			r_feedInCurrentLimit:= settings.Properties.r_ratedCurrentInput,
			r_supplyCurrentLimit:= settings.Properties.r_ratedCurrentInput,
			b_active := monitor.ACswitchgear.b_InputMCCBfb AND monitor.ACswitchgear.b_InputContactorfb AND b_InputACOK AND NOT b_gridTakeoverMode,
			b_enableSocTarget := b_SoCTargetEnable);


//Genset iso mode mapping (kind of peakshaver of genset)
	ePowerControlMode.PeakshaveInputGen:
		TargetData := MapGensetTarget(
				soft := control.SoftSettings.inputgenset,
				r_activePower := monitor.powermonitor.InputField.ar_ActivePower[0],
				r_reactivePower := monitor.powermonitor.InputField.ar_ReactivePower[0],
				r_Phasevoltage	:= monitor.powermonitor.InputField.ar_PhaseVoltage[0],
				b_active := monitor.ACswitchgear.b_InputMCCBfb AND monitor.ACswitchgear.b_InputContactorfb AND b_InputACOK,
				setpoints := gensetsetpoints);
	
		IF get.e_GensetMode = eGensetmode.FixedPower AND b_PSBactive THEN
			TargetData := MapGridTarget(
				slot1 := control.SoftSettings.PSB.setpointTimeslot1,
				slot2 := control.SoftSettings.PSB.setpointTimeslot2,
				r_activePower := monitor.peakshavebox.Powermonitor.ar_ActivePower,
				r_reactivePower := monitor.peakshavebox.Powermonitor.ar_ReactivePower,
				r_Phasevoltage	:= monitor.peakshavebox.Powermonitor.ar_PhaseVoltage[0],
				Peakshavemode := control.SoftSettings.PSB.PeakshaveMode,
				r_feedInCurrentLimit:= monitor.peakshavebox.r_MaxCTCurrent,
				r_supplyCurrentLimit:= monitor.peakshavebox.r_MaxCTCurrent,
				b_active := b_PSBActiveConditions AND SEL(control.softsettings.psb.b_BreakerControl,TRUE, monitor.peakshavebox.b_ContactorFb)
					AND NOT monitor.powerstack.b_InverterGridFormingMode
					AND monitor.powerstack.b_StartedState,
				b_enableSocTarget := b_SoCTargetEnable);
				b_SFCDeactivationEnable := control.softsettings.psb.b_BreakerControl;
		END_IF
END_CASE

//allow deactivation of powercontroller from inside functionblock
IF NOT b_SFCPIDActivation AND b_SFCDeactivationEnable THEN
	Targetdata.PIDmode := ePIDmode.None;
END_IF

//deload with PID controller
IF b_Deload THEN
	Targetdata.PIDmode := ePIDmode.BOTH;
	TargetData.r_FeedInCurrentLimit := 0;
	TargetData.r_SupplyCurrentLimit := 0;
	//TargetData.b_GenIsoPID := TRUE;
END_IF

//SOC drooping
IF (b_GridTakeOverMode OR eModeLocal = UgridIsland OR eModeLocal = UgridIso OR b_Deload) AND b_BESSReady THEN
	TargetData.b_EnableSocDrooping := FALSE;
ELSE
	TargetData.b_EnableSocDrooping := TRUE;
END_IF

//FUTURE WORK : make summation of multiple peakshave boxes.
END_METHOD

METHOD GetDiagnostics
VAR_IN_OUT
	AddError		: ARRAY [*] OF FB_AddErrorST;
	a_ActiveEvents	: ARRAY [*] OF ST_ErrorStruct;
	w_Index			: WORD;
END_VAR


VAR_INST
	s_dynamicStringModeTrans	: STRING := 'input disconnected by user, acknowledge to continue operation';;
	rTrigModeTrans				: R_TRIG;
END_VAR
(*Grid lost trip*)				AddError[w_Index](
		b_ErrorTrig				:= get.events.b_GridLostTrip,
		out_ST_Error			:= a_ActiveEvents[w_Index],
		w_ErrorID				:= 1,
		e_ObjectID				:= eObject_ID.GenGridController,
		s_Message				:= 'Grid loss trip',
		e_sev					:= eseverity.warning,
		b_autoClear				:= TRUE
	);
	w_Index := w_Index +1;
	
(**)	AddError[w_Index](
		b_ErrorTrig				:= FALSE,
		out_ST_Error			:= a_ActiveEvents[w_Index],
		w_ErrorID				:= 2,
		s_Message				:= '',
		e_sev					:= eseverity.info,
		b_autoClear				:= TRUE
	);
	w_Index := w_Index +1;
	
(**)		AddError[w_Index](
		b_ErrorTrig				:= FALSE,
		out_ST_Error			:= a_ActiveEvents[w_Index],
		w_ErrorID				:= 3,
		s_Message				:= '',
		e_sev					:= eseverity.info,
		b_autoClear				:= TRUE
	);
	w_Index := w_Index +1;
	

(*Over Freq Trip*)				AddError[w_Index](
		b_ErrorTrig				:= get.events.b_OverFreqTrip,
		out_ST_Error			:= a_ActiveEvents[w_Index],
		w_ErrorID				:= 4,
		s_Message				:= 'overfrequency trip',
		e_sev					:= eseverity.Warning,
	);
	w_Index := w_Index +1;
	
(*Under Freq Trip*)				AddError[w_Index](
		b_ErrorTrig				:= get.events.b_UnderFreqTrip,
		out_ST_Error			:= a_ActiveEvents[w_Index],
		w_ErrorID				:= 5,
		s_Message				:= 'underfrequency trip',
		e_sev					:= eseverity.Warning,
	
	);
	w_Index := w_Index +1;

(*Overload Trip*)			AddError[w_Index](
		b_ErrorTrig				:= get.events.b_OverloadTrip,
		out_ST_Error			:= a_ActiveEvents[w_Index],
		w_ErrorID				:= 6,
		s_Message				:= 'overload trip',
		e_sev					:= eseverity.Warning,
	);
	w_Index := w_Index +1;
	
(*SFC startup fault*)			AddError[w_Index](
		b_ErrorTrig				:= get.events.b_StartupFault,
		out_ST_Error			:= a_ActiveEvents[w_Index],
		w_ErrorID				:= 7,
		s_Message				:= 'Startup fault',
		e_sev					:= eseverity.Warning,
	);
	w_Index := w_Index +1;
	
(*SFC Sync fault*)			AddError[w_Index](
		b_ErrorTrig				:= get.events.b_SynchronisationFault,
		out_ST_Error			:= a_ActiveEvents[w_Index],
		w_ErrorID				:= 8,
		s_Message				:= 'Synchronisation fault',
		e_sev					:= eseverity.Warning,
	);
	w_Index := w_Index +1;

(*SFC warmup fault*)			AddError[w_Index](
		b_ErrorTrig				:= get.events.b_WarmupFault,
		out_ST_Error			:= a_ActiveEvents[w_Index],
		w_ErrorID				:= 9,
		s_Message				:= 'warmup fault',
		e_sev					:= eseverity.Warning,
	);
	w_Index := w_Index +1;
	
(*SFC shutdown timeout*)			AddError[w_Index](
		b_ErrorTrig				:= get.events.b_ShutdownTimeOut,
		out_ST_Error			:= a_ActiveEvents[w_Index],
		w_ErrorID				:= 10,
		s_Message				:= 'shutdown timeout',
		e_sev					:= eseverity.warning,
	);
	w_Index := w_Index +1;
	
(*breakermode transition iso inhibit*)			AddError[w_Index](
		b_ErrorTrig				:= get.events.b_TransToGenIsoInhibit,
		out_ST_Error			:= a_ActiveEvents[w_Index],
		w_ErrorID				:= 11,
		s_Message				:= 'generator iso mode inhibited, because grid ac was detected',
		e_sev					:= eseverity.warning,
		t_triggertime 			:= T#1S,
		b_autoclear				:= TRUE
	);
	w_Index := w_Index +1;
	
(*breakermode transition iso inhibit*)			AddError[w_Index](
		b_ErrorTrig				:= get.events.b_TransToGenDroopInhibit,
		out_ST_Error			:= a_ActiveEvents[w_Index],
		w_ErrorID				:= 12,
		s_Message				:= 'generator droop mode inhibited, because grid ac was detected',
		e_sev					:= eseverity.warning,
		t_triggertime 			:= T#1S,
		b_autoclear				:= TRUE
	);
	w_Index := w_Index +1;
	
	
	
	(*input grid active, acknowledge required*)			AddError[w_Index](
		b_ErrorTrig				:= get.events.b_TransFromInputGridAckRQ,
		out_ST_Error			:= a_ActiveEvents[w_Index],
		w_ErrorID				:= 13,
		s_Message				:= 'transition hold: input grid coupled, acknowledge by disconnecting AC or inputcontactor',
		e_sev					:= eseverity.warning,
		t_triggertime 			:= T#100MS,
		b_autoclear				:= TRUE
	);
	w_Index := w_Index +1;
	
rTrigModeTrans(CLK := get.b_ModeTransActive);
IF rTrigModeTrans.Q THEN
	IF get.events.b_CurrentLimitTrip THEN
		s_dynamicStringModeTrans := 'input disconnected by currentlimit trip, acknowledge to reconnect input';
	ELSIF get.events.b_EmstopDisconnect THEN
		s_dynamicStringModeTrans := 'input disconnected by EM-stop, clear EMstop and acknowledge to continue operation';
	ELSIF get.events.b_ShutdownDisconnect THEN
		s_dynamicStringModeTrans := 'input disconnected by shutdown, clear diagnostics and acknowledge to continue operation';
	ELSE
		s_dynamicStringModeTrans := 'input disconnected, acknowledge to continue operation';
	END_IF
END_IF
	
(*Mode transition active*)			AddError[w_Index](
		b_ErrorTrig				:= get.b_ModeTransActive,
		out_ST_Error			:= a_ActiveEvents[w_Index],
		w_ErrorID				:= 14,
		s_Message				:= s_dynamicStringModeTrans,
		e_sev					:= eseverity.warning,
		t_triggertime 			:= T#100MS,
		b_autoclear				:= TRUE
	);
	w_Index := w_Index +1;
	
(*input grid active, acknowledge required*)			AddError[w_Index](
		b_ErrorTrig				:= get.events.b_TransFromInputGenAckRQ,
		out_ST_Error			:= a_ActiveEvents[w_Index],
		w_ErrorID				:= 15,
		s_Message				:= 'transition hold: input genset started, acknowledge by stopping generator',
		e_sev					:= eseverity.warning,
		t_triggertime 			:= T#100MS,
		b_autoclear				:= TRUE
	);
	w_Index := w_Index +1;
	
(*genfix faulty start condition*)			AddError[w_Index](
		b_ErrorTrig				:= get.events.b_TransToGenFixInhibit,
		out_ST_Error			:= a_ActiveEvents[w_Index],
		w_ErrorID				:= 16,
		s_Message				:= 'AC detected at input before start stop was given, disconnect AC to continue',
		e_sev					:= eseverity.warning,
		t_triggertime 			:= T#100MS,
		b_autoclear				:= TRUE
	);
	w_Index := w_Index +1;
	
(*Starting inhibit*)			AddError[w_Index](
		b_ErrorTrig				:= get.events.b_StartingInhibit,
		out_ST_Error			:= a_ActiveEvents[w_Index],
		w_ErrorID				:= 17,
		s_Message				:= 'input control inhibited because input MCCB is opened',
		e_sev					:= eseverity.warning,
		t_triggertime 			:= T#100MS,
		b_autoclear				:= TRUE
	);
	w_Index := w_Index +1;
	
(*Starting inhibit*)			AddError[w_Index](
		b_ErrorTrig				:= get.events.b_RotationFieldFault,
		out_ST_Error			:= a_ActiveEvents[w_Index],
		w_ErrorID				:= 18,
		s_Message				:= 'Input rotation field fault, synchronization on hold',
		e_sev					:= eseverity.warning,
		t_triggertime 			:= T#100MS,
		b_autoclear				:= TRUE
	);
	w_Index := w_Index +1;
	
(*Gen down*)			AddError[w_Index](
		b_ErrorTrig				:= get.events.b_GenDownTrip,
		out_ST_Error			:= a_ActiveEvents[w_Index],
		w_ErrorID				:= 19,
		s_Message				:= 'Genset down trip, synchronization on hold',
		e_sev					:= eseverity.warning,
		t_triggertime 			:= T#100MS,
		b_autoclear				:= TRUE
	);
	w_Index := w_Index +1;
	
(*Overvoltage Trip*)			AddError[w_Index](
		b_ErrorTrig				:= get.events.b_OverVoltTrip,
		out_ST_Error			:= a_ActiveEvents[w_Index],
		w_ErrorID				:= 20,
		s_Message				:= 'overvoltage trip',
		e_sev					:= eseverity.Warning,
	);
	w_Index := w_Index +1;
	
(*Overvoltage Trip*)			AddError[w_Index](
		b_ErrorTrig				:= get.events.b_underVoltTrip,
		out_ST_Error			:= a_ActiveEvents[w_Index],
		w_ErrorID				:= 21,
		s_Message				:= 'undervoltage trip',
		e_sev					:= eseverity.Warning,
	);
	w_Index := w_Index +1;

(*Generator low fuel warning*)	AddError[w_Index](
		b_ErrorTrig				:= monitor.HartingIO.b_GenLowFuel,
		out_ST_Error			:= a_ActiveEvents[w_Index],
		w_ErrorID				:= 22,
		s_Message				:= 'Generator low fuel warning',
		e_sev					:= eseverity.Warning,
		b_autoclear				:= TRUE
	);
	w_Index := w_Index +1;
	
(*Generator Soc start warning*)	AddError[w_Index](
		b_ErrorTrig				:= monitor.battery.BatteryInfo.r_SOCScaled < GensetSetpoints.r_SocStart -1 AND SOCStart.Q,
		out_ST_Error			:= a_ActiveEvents[w_Index],
		w_ErrorID				:= 23,
		s_Message				:= 'autostart SoC low warning, Generator not started',
		e_sev					:= eseverity.warning,
		t_Triggertime			:= T#30S,
		b_autoclear				:= FALSE
	);
	w_Index := w_Index +1;
	
(*Generator Soc stop warning*)	AddError[w_Index](
		b_ErrorTrig				:= monitor.battery.BatteryInfo.r_SOCScaled > GensetSetpoints.r_SocStop +1 AND SOCStart.Q,
		out_ST_Error			:= a_ActiveEvents[w_Index],
		w_ErrorID				:= 24,
		s_Message				:= 'autostop SoC high warning, Generator power not stopped',
		e_sev					:= eseverity.Warning,
		t_Triggertime			:= T#30S,
		b_autoclear				:= FALSE
	);
	w_Index := w_Index +1;
END_METHOD

METHOD GridOkDetect : BOOL

VAR_INPUT
	SkipGridCode			: BOOL;
END_VAR

VAR_INST
	b_skip					: BOOL;
	tof_SyncDelay			: TOF := (PT := T#1S);
	
	ton_GridOK				: TON := (PT := T#2S);
	tof_GridLostBackup		: TOF ;
	ton_GCFaultReset		: Ton := (PT := T#60S);
	ton_FlatZeroPowerTimeOut: TON := (PT := T#1S);
	r_activepower			: REAL;
	GridCodeTripDetected	: BOOL;
END_VAR
tof_SyncDelay(IN := NOT b_breakerFB AND TargetData.Syncdata.b_Sync);
IF tof_syncDelay.Q THEN
	Settings.GridParams.ui_GCTripMaxTripTime := 500;
	
ELSE
	Settings.GridParams.ui_GCTripMaxTripTime := 40;
END_IF


tof_GridLostBackup(IN := b_BreakerACok, PT := TO_TIME(settings.GridParams.ui_GCTripMaxTripTime));


//detect flat power 
r_ActivePower := monitor.powermonitor.InputField.ar_ActivePower[0];
ton_FlatZeroPowerTimeOut(IN := r_ActivePower = 0 AND 
	b_breakerfb AND 
	ton_GridOK.Q AND monitor.powerstack.b_StartedState);

ton_GridOK(IN:= tof_GridLostBackup.Q);

b_skip := SkipGridcode OR NOT monitor.powerstack.b_StartedState OR b_gridtakeovermode;
ton_GCFaultReset(IN:= ton_GridOK.Q AND b_BreakerACok, PT := SEL(b_skip, TO_TIME(TO_REAL(settings.GridParams.ui_GCokReleaseTime)*1000), T#0S)); // AND ramp rate etc.etc. TBD

IF b_skip THEN
	b_GridCodeOK := ton_GridOK.Q;
ELSE
	b_GridCodeOK := ton_GCFaultReset.Q AND NOT b_GridCodeTripInverter AND NOT ton_FlatZeroPowerTimeOut.Q;
END_IF

get.events.b_GridLostTrip := NOT b_GridCodeOK;
GridOkDetect := b_gridCodeOK;
END_METHOD

ACTION IDLE_active:
get.e_state := eGenGridState.Idle;
b_SFCmodeTransInhibit := FALSE;
get.b_active := FALSE;

CASE breakerOperationMode OF
	ebreakeroperationmode.ExtGrid, ebreakeroperationmode.gridfeedthrough : b_ActivatePowerControl := FALSE;
	ELSE
		b_ActivatePowerControl := b_startcondition;
END_CASE
END_ACTION

ACTION INIT_active:
SFCResetTrigger := FALSE;

//Default init conditions
get.e_state := eGenGridState.Init;


CASE breakeroperationmode OF
	eBreakeroperationmode.Geniso, eBreakeroperationmode.GenDroop, eBreakeroperationmode.GenFix:
		b_IOstartStop := b_startcondition;
	eBreakerOperationMode.GridFeedthrough:
		GridOKdetect(TRUE);
END_CASE

IF BreakerOperationMode <> eBreakerOperationMode.ExtGrid THEN
	Extcontactor.Open(TRUE);	
END_IF

b_NetcontactorHoldClose := FALSE;
b_ActivatePowerControl := FALSE;
get.b_active := FALSE;
b_SFCmodeTransInhibit := FALSE;
//targetdata.Syncdata.b_Sync:= FALSE;
END_ACTION

METHOD InputContactorNC : BOOL
VAR_INPUT
	Enable 			: BOOL;
	//Toggle 		: BOOL;
END_VAR

VAR_INST
	TON_TriggerDelay 		: TON := (PT := T#500MS);
	TOF_ReleaseDelay 		: TOF := (PT := T#100MS);
	rtrig_ToggleState		: R_TRIG;
	rtrig_ToggleON			: R_TRIG;
	ftrig_ToggleOFF			: F_TRIG;
	b_ToggleState			: BOOL;
	ton_UpdateToggleState	: TON := (pt := T#500MS);
	b_Fb					: BOOL;
END_VAR
TON_TriggerDelay(IN := b_BreakerACOk AND Enable);
TOF_ReleaseDelay(IN:= TON_TriggerDelay.Q);
rtrig_ToggleON();
ftrig_ToggleOFF();	

IF get.b_ModeTransActive THEN
	b_ToggleState := FALSE;
	rtrig_ToggleON();
	ftrig_ToggleOFF.CLK := FALSE;
	rtrig_ToggleON.CLK := FALSE;
ELSE
	rtrig_ToggleON.CLK:= TON_TriggerDelay.Q;
	IF rtrig_ToggleON.Q THEN
		b_ToggleState := TRUE;
	END_IF
	
	ftrig_ToggleOFF(CLK := TOF_ReleaseDelay.Q);	
	IF ftrig_ToggleOFF.Q THEN
		b_ToggleState := FALSE;
	END_IF
END_IF


IF b_ToggleState THEN
	b_Fb := InputContactor.Close(TRUE);
ELSE
	b_Fb := NOT InputContactor.open(TRUE);
END_IF
END_METHOD

METHOD MapGensetTarget : ST_PowerControl_Target
VAR_IN_OUT CONSTANT
	soft		: ST_SoftSettings_Genset;
END_VAR

VAR_IN_OUT
	setpoints 	: ST_Genset_setpoints;
END_VAR

VAR_INPUT
	r_ActivePower				: REAL;
	r_ReactivePower				: REAL;
	r_phaseVoltage				: REAL;
	b_active					: BOOL;
END_VAR


VAR_INST
	r_chargePowerTarget			: REAL := 100; 
	r_GensetMaxCurrent			: REAL;
	r_GensetMinPower			: REAL;
	r_GensetMinCurrent			: REAL;
	r_GensetEffPower			: REAL;
	r_GensetEffCurrent			: REAL;
	r_GenCurSetpointModified	: REAL;
	r_GenCurSetpointLoadStart	: REAL;
	r_GenCurSetpointTemp		: REAL;
	r_GenCurSetpoint			: REAL;
	r_loadbankMaxCurrent		: REAL;
	enable						: BOOL := TRUE;
	r_dischargeloadmax			: REAL := 100;
	r_Chargeloadmax				: REAL := 100;
	r_loadmaxActual				: REAL;
	r_RatedInputCurrent			: REAL;
	ton_GenMaxCurrentDelay		: TON := (PT := T#5S);
	
	b_ConditionalStart			: BOOL;
	
	//params
	by_genloadMinLimit			: BYTE := 5;
END_VAR
IF b_TimeSlot2 THEN
	setpoints := soft.setpointTimeslot2;
ELSE 
	setpoints := soft.setpointTimeslot1;
END_IF

MapgensetTarget.r_PIDRampRate := soft.Generator.r_ramprate;
MapgensetTarget.b_GenIsoPID  := FALSE; 
MapGensetTarget.PeakshaveMode := FALSE;
r_RatedInputCurrent := settings.Properties.r_ratedCurrentInput;
r_chargePowerTarget := settings.Properties.r_RatedActivePower;

IF st_params.GenIso_InverterMode = eGenIsoInverterMode.ISO_SLOWDROOP AND soft.generator.e_GensetMode = egensetmode.Isochronous THEN
	MapgensetTarget.r_droopMinimum := 20;
ELSE
	MapgensetTarget.r_droopMinimum := 0.1;
END_IF

//calculate related values from genset settings
r_GensetMaxCurrent := LIMIT(0, ABS(KWtoCurrent(soft.Generator.r_RatedPower * soft.Generator.r_powerloadMax / 100, r_phaseVoltage * 1.73)), r_RatedInputCurrent);
r_GensetMinCurrent := LIMIT(by_genloadMinLimit, ABS(KWtoCurrent(soft.Generator.r_RatedPower * soft.Generator.r_powerloadMin / 100, r_phaseVoltage * 1.73)), r_RatedInputCurrent);
r_GensetEffPower := soft.Generator.r_RatedPower * soft.Generator.r_powerloadEff / 100;
r_GensetEffCurrent := LIMIT(0, ABS(KWtoCurrent(r_GensetEffPower, r_phaseVoltage * 1.73)), r_RatedInputCurrent);
r_loadbankMaxCurrent := LIMIT(0, ABS(KWtoCurrent(soft.Loadbank.r_PowerRating, r_phaseVoltage * 1.73)), r_RatedInputCurrent);
r_dischargeloadmax := MIN(monitor.powerstack.r_Pmax / MAX(1, monitor.powerstack.r_RatedPower) * 100, 100);
r_Chargeloadmax := -MIN(monitor.powerstack.r_Pmin / MAX(1, monitor.powerstack.r_RatedPower) * 100, 100);

r_loadmaxActual := MAX(setpoints.r_BatteryloadStart, r_DisChargeloadmax);


//shift setpoint from eff. to max point if battery is at limit.
IF monitor.powerstack.e_PowerState = ePowerstate.Charging THEN
	r_GenCurSetpointLoadStart := r_GensetEffCurrent;
ELSE
	r_GenCurSetpointLoadStart := scale(
	monitor.powerstack.r_Loadpercent, 
	r_loadmaxActual - 3, 
	r_loadmaxActual,
	r_GensetEffCurrent,
	r_GensetMaxCurrent);
END_IF

b_ConditionalStart := (LoadStart.Q OR SOCStart.Q OR BatFullStart.Q OR ChargeLoadStart.Q);

ton_GenMaxCurrentDelay(IN:= b_ConditionalStart AND MAX(0, Monitor.powermonitor.OutputField.ar_ActivePower[0] + r_chargePowerTarget) > r_GensetEffPower);
IF ton_GenMaxCurrentDelay.Q THEN
	r_GenCurSetpointModified := r_GensetMaxCurrent;
ELSIF NOT b_ConditionalStart THEN
	r_GenCurSetpointModified := r_gensetMinCurrent;
ELSE 
	r_GenCurSetpointModified := r_GenCurSetpointLoadStart;
END_IF
	
//shift setpoint from current to zero if generator can not maintain frequency.
IF soft.generator.e_GensetMode = egensetmode.Isochronous AND emodelocal <> UgridDroop THEN
	r_GenCurSetpoint := LIMIT(0,scale(
		monitor.powerstack.r_FrequencyD7,
		settings.GridParams.r_GridFrequencyMin, 
		monitor.controlfb.Operation.system.r_NominalFrequency,
		0,
		r_GenCurSetpointModified),
		r_GenCurSetpointModified);
ELSE
	r_GenCurSetpoint := r_GenCurSetpointModified;	
END_IF

//Iso generator power setpoint override by user
IF monitor.controlfb.Operation.system.r_Pset < 0 THEN
	r_GenCurSetpoint := kwtoCurrent(-monitor.controlfb.Operation.system.r_Pset, monitor.powermonitor.OutputField.ar_LineVoltage[0]);
END_IF


//Activate mode
IF b_active AND (b_TimeSlot1 OR b_TimeSlot2) AND enable THEN
	CASE soft.generator.e_GensetMode OF
		egensetmode.FixedPower:
			MapGensetTarget.PIDmode := ePIDmode.None;
//		egensetmode.Droop:
//			MapgensetTarget.b_DisableSocDrooping := FALSE;
//			MapGensetTarget.r_FeedInCurrentLimit := settings.Properties.r_ratedCurrentInput;
//			MapGensetTarget.r_SupplyCurrentLimit := settings.Properties.r_ratedCurrentInput;
//			MapGensetTarget.PIDmode := ePIDmode.None;
		egensetmode.Isochronous, egensetmode.Droop:
			MapgensetTarget.b_GenIsoPID := TRUE;
			MapGensetTarget.r_SupplyCurrentLimit := MIN(r_gencursetpoint, settings.Properties.r_ratedCurrentInput);
			MapGensetTarget.r_FeedInCurrentLimit := -  MIN(r_gencursetpoint, settings.Properties.r_ratedCurrentInput);
			MapGensetTarget.PIDmode := ePIDmode.BOTH;
	END_CASE
END_IF

//raise invalid params and disable PID
IF r_GensetMinCurrent > r_GensetEffCurrent OR r_GensetEffCurrent > r_GensetMaxCurrent THEN
	get.events.b_InvalidGensetParameters := TRUE;
ELSE
	get.events.b_InvalidGensetParameters := FALSE;
END_IF

//reset current limits, to have nice ramp when starting.
IF MapGensetTarget.PIDmode = ePIDmode.None THEN
	MapGensetTarget.r_FeedInCurrentLimit := -r_GensetMinCurrent;
	MapGensetTarget.r_SupplyCurrentLimit := r_GensetMinCurrent;
END_IF

//Loadbank control, overwrite existing targetvalues
IF batfullstart.Q OR ChargeLoadStart.Q THEN
	MapGensetTarget.r_FeedInCurrentLimit := r_loadbankMaxCurrent;
	MapGensetTarget.r_SupplyCurrentLimit := 0;
END_IF

MapGensetTarget.Measurements.r_ActivePower := r_ActivePower;		
MapGensetTarget.Measurements.r_PhaseVoltage := r_PhaseVoltage;
MapGensetTarget.Measurements.r_ReactivePower:= r_ReactivePower;
END_METHOD

METHOD MapGridTarget : ST_PowerControl_Target;
VAR_IN_OUT CONSTANT
	Slot1 						: ST_peakshave_setpoints;
	Slot2 						: ST_peakshave_setpoints;
	r_ActivePower				: ARRAY [0..3] OF REAL;
	r_ReactivePower				: ARRAY [0..3] OF REAL;
END_VAR

VAR_INST
	b_enable: BOOL;
	singlePhaseMode : BOOL;
	
	sr_socTarget	: SR;
	r_IdlePowerTarget : REAL;
	r_SocTarget	: REAL;
END_VAR

VAR_INPUT
	r_phaseVoltage				: REAL;
	r_FeedInCurrentLimit		: REAL;
	r_SupplyCurrentLimit		: REAL;
	b_active					: BOOL;
	b_enableSocTarget			: BOOL;
	PeakshaveMode				: ePeakshaveMode;
END_VAR

VAR
	i_reverseFactor				: INT;
END_VAR
//define value which is invalid such that function will not be used.
MapgridTarget.r_PIDRampRate := settings.MachineParams.system.GenGridController.r_PIDLimitRampDefault;
MapgridTarget.b_GenIsoPID := FALSE;	
MapGridtarget.PeakshaveMode := TRUE;

b_enable :=  b_active AND (b_TimeSlot1 OR b_TimeSlot2);

MapGridTarget.r_FeedInCurrentLimit := ThreepointSelector(
		r1max := r_FeedinCurrentLimit,
		r2 := slot1.r_FeedInCurrentLimitSoft,
		r3 := slot2.r_FeedInCurrentLimitSoft,
		b2 := b_TimeSlot1,
		b3 := b_TimeSlot2);
		
	MapGridTarget.r_SupplyCurrentLimit := ThreepointSelector(
		r1max := r_SupplyCurrentLimit,
		r2 := slot1.r_SupplyCurrentLimitSoft,
		r3 := slot2.r_SupplyCurrentLimitSoft,
		b2 := b_TimeSlot1,
		b3 := b_TimeSlot2);

	r_IdlePowerTarget := ThreepointSelector(
		r1max := 1000,
		r2 := slot1.r_IdleChargePower,
		r3 := slot2.r_IdleChargePower,
		b2 := b_TimeSlot1,
		b3 := b_TimeSlot2);
		
	r_SocTarget := ThreepointSelector(
		r1max := 100,
		r2 := slot1.r_SocTarget,
		r3 := slot2.r_SocTarget,
		b2 := b_TimeSlot1,
		b3 := b_TimeSlot2);
		
IF b_enable THEN
	MapGridTarget.PIDmode := ePIDmode.Both;
	
	
	IF b_enableSocTarget THEN
		sr_socTarget(
			SET1 := r_soc < r_SocTarget - st_params.r_SocHysteresis OR r_soc > r_SocTarget + st_params.r_SocHysteresis,
			RESET := r_soc = r_soctarget);
		
		IF r_Soc < r_socTarget AND sr_socTarget.Q1 THEN // when idletarget set to charging (negative) or soc target implies charging
			MapGridTarget.r_PowerTarget := -r_IdlePowerTarget;
		ELSIF r_Soc > r_SocTarget AND sr_socTarget.Q1 THEN
			MapGridTarget.r_PowerTarget := r_IdlePowerTarget;
		ELSE
			MapGridTarget.r_PowerTarget := 0;
		END_IF
	ELSE
		MapGridTarget.r_PowerTarget := control.Operation.system.r_Pset;	
	END_IF

ELSE
	//MapGridTarget.r_FeedInCurrentLimit := monitor.powerstack.r_RatedPower;
	//MapGridTarget.r_SupplyCurrentLimit := monitor.powerstack.r_RatedPower;
	MapGridTarget.PIDmode := ePIDmode.None;
END_IF

PeakshaveTotalizer(
	ActivePower := r_ActivePower,
	ReactivePower := r_ReactivePower,
	FeedInCurrent_A := MapGridTarget.r_FeedInCurrentLimit,
	SupplyCurrent_A := MapGridTarget.r_SupplyCurrentLimit,
	singleMode := PeakshaveMode = ePeakshaveMode.Singlephase,
	PhaseVoltage_V := r_phaseVoltage,
	TotalActivePowerMod => MapGridTarget.Measurements.r_ActivePower,
	TotalReactivePowerMod => MapGridTarget.Measurements.r_ReactivePower);

MapGridTarget.Measurements.r_PhaseVoltage := r_PhaseVoltage;
END_METHOD

METHOD PRIVATE ModeSwitch : BOOL
VAR_INPUT
	RequestedMode			: eBreakerOperationMode;
END_VAR

VAR_INST
	b_EnableInputGridTriggers	: BOOL;
	b_ManualinputControl	: BOOL;
	rTrigModeTransManualClose	: R_TRIG;
	rTrigModeTransToggle		: R_TRIG;
	rTrigModeTransEmstop		: R_TRIG;
	fTrigReset					: F_TRIG;
	rTrigModeTransshutdown		: R_TRIG;
	rTrigModeTransCLimit		: R_TRIG;
	fTrigModeACreleased			: F_TRIG;
	tofRetryTimeOut				: TOF := (PT := T#60S);
	by_cLimitCounter			: BYTE;
	AllowModeSwitch				: BOOL;
	b_inhibitSum				: BOOL;
	b_AckRQSum					: BOOL;
	b_allowModeTransGen			: BOOL;
	
	b_GridAtOutput				: BOOL;
	b_UnwantedGenACatInput		: BOOL;	
	
	TonRecoverFromDisconnectDelay	: TON := (PT:= T#1S);
END_VAR
//reset events
get.events.b_TransToGenDroopInhibit := FALSE;
b_ManualinputControl := FALSE;
b_EnableInputGridTriggers := FALSE;
get.events.b_TransToGenIsoInhibit := FALSE;
get.events.b_TransToGenFixInhibit := FALSE;
get.events.b_TransFromInputGridAckRQ := FALSE;
get.events.b_TransFromInputGenAckRQ := FALSE;
b_allowModeTransGen := FALSE;
get.events.b_StartingInhibit := NOT b_InputMCCBfb AND BreakerOperationMode <> eBreakerOperationMode.None;
//Predefine some conditions
b_GridAtOutput := monitor.powerstack.b_GridACdetected AND NOT inputcontactor.b_fb AND NOT monitor.powerstack.b_InverterGridFormingMode;
b_UnwantedGenACatInput := b_inputACOK AND NOT inputcontactor.b_fb AND b_BusbarACOK;
get.b_ModeChanged := RequestedMode <> BreakerOperationMode;


//inhibited conditions
CASE RequestedMode OF
	eBreakerOperationMode.GenIso: 
		get.events.b_TransToGenIsoInhibit := b_GridAtOutput OR b_AFEactive;
	eBreakerOperationMode.GenDroop:
		get.events.b_TransToGenDroopInhibit := b_GridAtOutput OR b_AFEactive; // OR b_UnwantedGenACatInput;
	eBreakerOperationMode.genfix:
		get.events.b_TransToGenFixInhibit := b_UnwantedGenACatInput;
END_CASE

fTrigModeACreleased();
//Acknowledgeable conditions
CASE BreakerOperationMode OF
	eBreakerOperationMode.GridFeedthrough: 
		b_EnableInputGridTriggers := TRUE;
		b_ManualinputControl	:= NOT (b_autoSwitching OR b_Breakerfb OR get.b_ModeChanged);
		fTrigModeACreleased.CLK := b_breakerACOK;
		get.events.b_TransFromInputGridAckRQ := RequestedMode <> BreakerOperationMode AND InputContactor.b_fb AND b_inputACOK;
	eBreakerOperationMode.GenDroop, eBreakerOperationMode.GenIso: 
		get.events.b_TransFromInputGenAckRQ := RequestedMode <> BreakerOperationMode AND ((InputContactor.b_fb AND b_inputACOK) OR b_IOStartStop) AND enable;
		IF RequestedMode = eBreakerOperationMode.GenIso OR RequestedMode = eBreakerOperationMode.GenDroop THEN
			get.events.b_TransFromInputGenAckRQ := FALSE;
			b_allowModeTransGen := TRUE;
		END_IF
		
		b_SkipGensetCooldown := RequestedMode = eBreakerOperationMode.GridFeedthrough;
END_CASE

b_AckRQSum := 
	get.events.b_TransFromInputGridAckRQ OR
	get.events.b_TransFromInputGenAckRQ OR b_ManualinputControl;

b_inhibitSum := 
	get.events.b_TransToGenIsoInhibit OR
	get.events.b_TransToGenDroopInhibit OR
	b_SFCmodeTransInhibit;

IF BreakerOperationMode = RequestedMode AND NOT b_inhibitSum THEN
	get.b_ModeTransInhibit := FALSE;
ELSE
	get.b_ModeTransInhibit := b_inhibitSum;
END_IF

get.b_ShowModeTrans := ShowModeTransButton();

//if SFC is not active
IF NOT get.b_active THEN
	AllowModeSwitch := NOT (get.b_ModeTransInhibit OR b_AckRQSum);
ELSE
	AllowModeSwitch := b_allowModeTransGen;	
END_IF

//MODE CHANGE TRIGGERS
rTrigModeTransClimit(
	CLK := CurrentLimitProtection(
				enable := control.SoftSettings.inputgrid.Breaker.CurrentLimitDisconnect AND b_EnableInputGridTriggers,
				FeedinLimit := targetdata.r_FeedInCurrentLimit,
				SupplyLimit := targetdata.r_SupplyCurrentLimit,
				Current := monitor.powermonitor.InputField.ar_Current[0],
				power := monitor.powermonitor.inputfield.ar_activepower[0],
				tripdelay := st_params.CurrentLimitTripDelay));

// reset counter after 1 min of the trigger event.
tofRetryTimeOut(IN := rTrigModeTransClimit.Q);
IF NOT tofRetryTimeOut.Q THEN
	by_cLimitCounter := 0;
END_IF
		
IF rTrigModeTransClimit.Q THEN
	by_cLimitCounter := by_cLimitCounter + 1;
	get.events.b_CurrentLimitDisconnect := TRUE;
	get.b_ModeTransActive := TRUE;
END_IF

IF by_climitCounter > 0 AND get.b_ModeTransActive AND NOT b_breakerfb THEN
	get.events.b_CurrentLimitDisconnect := FALSE;
	IF by_climitCounter <= control.SoftSettings.inputgrid.Breaker.CurrentLimitRetries THEN
		get.b_ModeTransActive := FALSE;
	ELSE
		get.events.b_CurrentLimitTrip := TRUE;
	END_IF
END_IF

TonRecoverFromDisconnectDelay();
// triggers for disconnection of input
IF b_EnableInputGridTriggers AND settings.Configuration.b_ACInputConnection THEN
	rTrigModeTransEmstop(CLK := (gvl.b_QuickshutdownActive OR gvl.b_EmergencyShutdownActive) AND control.SoftSettings.inputgrid.Breaker.EMstopDisconnect);
	IF rTrigModeTransEmstop.Q THEN get.events.b_EmstopDisconnect := TRUE; TonRecoverFromDisconnectDelay.IN := b_autoSwitching; get.b_ModeTransActive := TRUE; END_IF
	rTrigModeTransShutdown(CLK := Monitor.system.e_State = eSystemState.shutdown AND control.SoftSettings.inputgrid.Breaker.ShutdownDisconnect);
	IF rTrigModeTransShutdown.Q THEN  get.events.b_shutdownDisconnect := TRUE; TonRecoverFromDisconnectDelay.IN := b_autoSwitching; get.b_ModeTransActive := TRUE; END_IF
	rTrigModeTransToggle(CLK := b_ActivateTransition);
	IF rTrigModeTransToggle.Q THEN get.b_ModeTransActive := NOT get.b_ModeTransActive; END_IF
	rTrigModeTransManualClose(CLK := b_ManualinputControl);
	IF rTrigModeTransManualClose.Q THEN get.b_ModeTransActive := TRUE; TonRecoverFromDisconnectDelay.IN := FALSE; END_IF
ELSE
	get.b_ModeTransActive := FALSE;	
END_IF

//auto clear emstop trigger once battery is ready again after EMstop
IF TonRecoverFromDisconnectDelay.Q AND b_BESSReady AND get.b_ModeTransActive THEN
	TonRecoverFromDisconnectDelay.IN := FALSE;
	get.b_ModeTransActive := FALSE;
END_IF

//reset disconnection triggers
fTrigReset(CLK := get.b_ModeTransActive);
IF fTrigReset.Q THEN
	get.events.b_EmstopDisconnect := FALSE;
	get.events.b_ShutdownDisconnect := FALSE;
END_IF

ModeSwitch := AllowModeSwitch AND NOT get.b_ModeTransActive;
END_METHOD

METHOD PeakshaveTotalizer : BOOL
(*
    PeakshaveTotalizer
    - Inputs:
        ActivePower[kW], ReactivePower[kvar] per phase; index 0 = totals
        FeedInCurrent_A (>=0), SupplyCurrent_A (>=0)  -- CURRENT limits
        SingleMode = TRUE  -> enforce per-phase envelope (recommended)
        SingleMode = FALSE -> pass-through totals (with optional slew)
        PhaseVoltage_V = L-N RMS (e.g. 230 V)
        SafetyMargin_kW : small guard so we don't graze the boundary
        EnvTau_s        : low-pass on the safe envelope to kill jitter
        SlewP_kW_per_s / SlewQ_kvar_per_s with CycleTime_s
    - Outputs:
        TotalActivePowerMod (kW), TotalReactivePowerMod (kvar)
*)

VAR_IN_OUT CONSTANT
    ActivePower   : ARRAY[0..3] OF REAL;   // kW   [0]=totaal, [1..3]=L1..L3
    ReactivePower : ARRAY[0..3] OF REAL;   // kvar [0]=totaal, [1..3]=L1..L3
END_VAR
VAR_INPUT
    FeedInCurrent_A  : REAL;               // per-fase exportlimiet [A]
    SupplyCurrent_A  : REAL;               // per-fase importlimiet [A]
    SingleMode       : BOOL;               // TRUE = fase-selectie
    PhaseVoltage_V   : REAL := 230.0;      // L-N spanning [V]
END_VAR
VAR_OUTPUT
    TotalActivePowerMod   : REAL;          // kW
    TotalReactivePowerMod : REAL;          // kvar
END_VAR
VAR_INST
    Vph : REAL;
    Ptot, Qtot : REAL;
    Pmod: REAL;
    tmp : REAL;
END_VAR
(* basis: LN spanning *)
IF PhaseVoltage_V > 0.0 THEN
    Vph := PhaseVoltage_V;
ELSE
    Vph := 230.0;
END_IF;

Ptot := ActivePower[0];
Qtot := ReactivePower[0];

(* Multiphase = gewoon totaal doorgeven *)
IF NOT SingleMode THEN
    TotalActivePowerMod   := Ptot;
    TotalReactivePowerMod := Qtot;
    PeakshaveTotalizer := TRUE;
    RETURN;
END_IF;

(* kandidaat totaal = 3 × fase *)
Ptot := ActivePower[0];
IF Ptot > 30 THEN
    Pmod := 3.0 * MAX(ActivePower[1], ActivePower[2], ActivePower[3]);   // export: hoogste fase ×3
ELSIF Ptot < 0 THEN
    Pmod := 3.0 * MIN(ActivePower[1], ActivePower[2], ActivePower[3]);   // import: laagste (meest neg.) fase ×3
ELSE
    Pmod := Ptot;          // of ActivePower[0], of een kleine deadband
END_IF

(* kandidaat totaal = 3 × fase *)
//Pmod := 3.0 * ActivePower[phase];

(* outputs *)
TotalActivePowerMod   := Pmod;   // hierop laat je PID peakshaven
TotalReactivePowerMod := Qtot;   // Q onveranderd
PeakshaveTotalizer := TRUE;
END_METHOD

METHOD Reset : BOOL
VAR_INPUT
END_VAR

VAR_INST
	EmptyEventStruct 	: ST_GengridController_events;
END_VAR
get.events := EmptyEventStruct;
RESET := GenFreqVoltProtections(FALSE, FALSE ,TRUE, 0);
END_METHOD

ACTION RUN_active:
get.e_state := eGenGridState.Running;
SFCTransTrigger.in := FALSE;

//TRANSITION
CASE BreakerOperationMode OF
	eBreakerOperationMode.GenIso, eBreakerOperationMode.GenDroop:
		b_ActivatePowerControl := b_GenStarted;
		get.b_gensetStarting := FALSE;
		IF b_hybridMode THEN
			SFCTransTrigger.in := GenDownCheck(TRUE, FALSE);
		ELSE
			SFCTransTrigger.in := NOT b_StartCondition OR GenDownCheck(TRUE, FALSE);
		END_IF
		
		
	eBreakerOperationMode.Genfix:
		//SFCTransTrigger.in := NOT b_StartCondition OR GenDownCheck(TRUE, FALSE)  OR GenFreqProtections(TRUE, FALSE,FALSE, Monitor.powermonitor.InputField.ar_ActivePower[0]);
		//SFCTransTrigger.in := GenDownCheck(b_StartCondition, FALSE) OR GenFreqProtections(TRUE, FALSE,FALSE, Monitor.powermonitor.InputField.ar_ActivePower[0]);
		SFCTransTrigger.in := NOT b_BusbarACOK OR GenFreqVoltProtections(TRUE, FALSE,FALSE, Monitor.powermonitor.InputField.ar_ActivePower[0]);
		b_IOstartStop := b_StartCondition;
		get.b_gensetStarting := FALSE;
		b_ActivatePowerControl := b_GenStarted;
		IF NOT b_IOstartStop THEN
			get.e_state := eGenGridState.Waiting_Trigger;
		ELSE
			IF Monitor.powermonitor.InputField.ar_ActivePower[0] = 0 THEN
				get.e_state := eGenGridState.Starting;
			END_IF
		END_IF
	
	eBreakerOperationMode.GridFeedthrough, eBreakerOperationMode.ExtGrid: 
		b_ActivatePowerControl := TRUE;
		IF NOT GridOKDetect(NOT b_AMFEnabled) OR ZeroCurrentDisconnect() THEN
			IF NOT b_AutoSwitching THEN
				Get.b_ModeTransActive := TRUE;
			ELSE
				SFCTransTrigger.in := TRUE;
			END_IF
		END_IF
END_CASE

IF NOT monitor.powerstack.b_ControlEnabled OR NOT b_breakerfb OR Get.b_ModeTransActive OR NOT b_InputMCCBfb THEN
	SFCTransTrigger.in := TRUE;
END_IF

SFCtip := SFCTransTrigger.Q AND NOT SFCtip;
END_ACTION

METHOD SetBreakerAndPowercontrolMode : BOOL
VAR_INPUT
	ACInputType				: eACinputType;
	GridMode				: eGridMode;
	GensetMode				: eGensetMode;
	PSBMode					: ePSBMode;
	//b_extBreakerControl		: BOOL;
	PSBenable				: BOOL;
	b_extGenset				: BOOL;
END_VAR

VAR_IN_OUT
	PowerControlMode		: ePowerControlMode;
	ExtGensetMode			: BOOL;
END_VAR

VAR_INST
	RequestedBreakerMode	: eBreakerOperationMode;
END_VAR
//Initialize values
get.events.b_TransToGenIsoInhibit := FALSE;


	

//Default values
RequestedBreakerMode := eBreakerOperationMode.none;
CASE ACInputType OF
	eACinputType.grid: 
		RequestedBreakerMode := eBreakerOperationMode.GridFeedthrough;
	eACinputType.Genset: 
		CASE GensetMode OF
			eGensetMode.isochronous				: RequestedBreakerMode := eBreakerOperationMode.GenIso;
			eGensetMode.Droop					: RequestedBreakerMode := eBreakerOperationMode.GenDroop;
			eGensetMode.FixedPower				: RequestedBreakerMode := eBreakerOperationMode.GenFix;
		END_CASE
END_CASE

//breaker mode is most strict, and can be changed if modetransinhibit and no transition is active. ==> output of method
IF Modeswitch(RequestedMode := RequestedBreakerMode) THEN
	BreakerOperationMode := RequestedBreakerMode;	
END_IF

//power control is less strict, and can be changed if modetransinhibit is false
IF NOT get.b_ModeTransInhibit AND BreakerOperationMode = RequestedBreakerMode THEN
	CASE ACInputType OF
		eACinputType.grid: 
			PowerControlMode := ePowerControlMode.PeakshaveInputGrid; 
		eACinputType.Genset: 
			PowerControlMode := ePowerControlMode.PeakshaveInputGen;
		eACinputType.None:
			PowerControlMode:= ePowerControlMode.none;	
	END_CASE
END_IF


// Activation of PSB as powercontrol source (only when no generator is at input)
IF PSBenable AND BreakerOperationMode < 3 THEN
	CASE PSBMode OF
		ePSBMode.Monitor:
			PowerControlMode:= ePowerControlMode.PeakshaveExt;
		ePSBMode.MonitorControl:
			RequestedBreakerMode := eBreakerOperationMode.ExtGrid;		
	END_CASE
END_IF

	//ext genset control enabling
ExtGensetMode := ACInputType <> eACinputType.Genset AND b_extGenset;
get.b_gensetcontrol:= b_extGenset OR BreakerOperationMode = eBreakerOperationMode.GenFix OR BreakerOperationMode = eBreakerOperationMode.GenIso; 

//Fill get 
get.e_BreakerMode := BreakerOperationMode;
get.e_PowerControlMode := PowerControlMode;
get.e_GensetMode := control.softSettings.inputgenset.generator.e_GensetMode;
get.b_extGensetMode := ExtGensetMode;
END_METHOD

METHOD SetInverterMode : BOOL
VAR_INPUT
	Gridmode			: 	eGridmode;
	UgridPowermode		: 	eUgridpowermode;
	BreakerMode			:	eBreakerOperationMode;
	PSBMode				: 	ePSBMode;
	b_InputGridcodeEnabled	: 	BOOL;
	b_gridacDetected	: 	BOOL;
	b_PowerstackStarted	:	BOOL;
	b_ExtFb				: 	BOOL; //OPEN IS TRUE
	b_InputFB			: 	BOOL; //OPEN IS TRUE
	b_AMF				: 	BOOL;
END_VAR

VAR_OUTPUT
	b_MasterSlaveEnabled: BOOL;
END_VAR

VAR_INST
	b_parallelUgrid		: 	BOOL;
	b_test : BOOL;
END_VAR
b_ExtGridConnected := FALSE;
b_slowLom := TRUE;


//Get invertermode from breakermode
CASE BreakerMode OF
	eBreakerOperationMode.none:
		IF inputcontactor.b_fb THEN
			InputContactor.open(TRUE);
		END_IF
		b_slowLom := FALSE;
		
		IF NOT b_PowerstackStarted THEN
			IF NOT b_gridAcDetected THEN
				eModeLocal := UgridIsland;
			ELSE
				eModeLocal := AFE;
			END_IF
		END_IF
		
		//Overwrite for manual choice user or overruling parameters
	CASE gridmode OF
		egridmode.following: eModeLocal := AFE;
		egridmode.forming: eModeLocal := UgridDroop;	
	END_CASE
		
	eBreakerOperationMode.GridFeedthrough:
		IF NOT get.b_active AND NOT monitor.powerstack.b_ControlEnabled THEN
			InputContactorNC(b_autoSwitching);
		END_IF
		
		b_ExtGridConnected := b_inputACOK AND b_InputFB;
		IF NOT b_InputFB AND (NOT b_gridACdetected OR Gridmode = eGridmode.forming) THEN // OR (NOT b_netcontactorFB AND NOT GridOKdetect(FALSE)) THEN
			eModeLocal := SEL(Gridmode = eGridmode.forming, UgridIsland, UgridDroop);
		ELSIF b_inputgridCodeEnabled AND Gridmode <> egridmode.forming AND NOT get.b_ModeTransActive THEN
			eModeLocal := AFE;
		ELSE
			eModeLocal := UgridIso;
			b_slowLom := control.SoftSettings.inputgrid.b_WeakGridInput AND NOT b_inputgridCodeEnabled;
		END_IF
			
	eBreakerOperationMode.GenDroop:
		IF NOT get.b_active AND NOT monitor.powerstack.b_ControlEnabled AND NOT get.b_ModeTransActive THEN
			IF get.e_GensetStartStop = eGensetStartStop.Start AND monitor.ACswitchgear.b_InputMCCBfb THEN
					Inputcontactor.Close(TRUE);
			ELSE
					Inputcontactor.Open(TRUE);
			END_IF
		END_IF
		eModeLocal := UgridDroop;
	
	eBreakerOperationMode.GenFix:
		IF NOT get.b_active AND NOT monitor.powerstack.b_ControlEnabled AND NOT get.b_ModeTransActive THEN
			IF get.e_GensetStartStop = eGensetStartStop.Start AND monitor.ACswitchgear.b_InputMCCBfb THEN
					Inputcontactor.Close(TRUE);
			ELSIF NOT b_BusbarACOK THEN
				 Inputcontactor.Open(TRUE);		
			END_IF
		END_IF
	
		eModeLocal := UgridIsland;
		IF b_gridAcDetected THEN
			eModeLocal := AFE;
		END_IF
		
	eBreakerOperationMode.GenIso:
		b_slowLom := TRUE;
		IF NOT get.b_active AND NOT monitor.powerstack.b_ControlEnabled AND NOT get.b_ModeTransActive THEN
			IF get.e_GensetStartStop = eGensetStartStop.Start AND monitor.ACswitchgear.b_InputMCCBfb THEN
					Inputcontactor.Close(TRUE);
			ELSE
					Inputcontactor.Open(TRUE);
			END_IF
		END_IF
		
		IF st_params.GenIso_InverterMode <> eGenIsoInvertermode.AFE THEN
			eModeLocal := UgridIso;
		ELSE
			eModeLocal := AFE;
		END_IF
	
		IF NOT b_InputFB THEN
			eModeLocal := SEL(Gridmode = eGridmode.forming, UgridIsland, UgridDroop);
		END_IF
		
	eBreakerOperationMode.ExtGrid:
		eModeLocal := AFE;
		IF b_AMF AND b_ExtFb THEN
			eModeLocal := UgridIsland;
		END_IF
END_CASE

//Overwrite for grid detection
//IF b_AcDetected THEN
//	eModeLocal := AFE;
//END_IF

CASE GridMode OF
	eGridmode.forming: 
		eModeLocal := UgridDroop;
	eGridmode.following: 
		eModeLocal := AFE;	
END_CASE

//Catch mode inverter and powermode
CASE eModeLocal OF
	AFE 		: InverterMode := eInverterModes.Afe; PowerMode :=  ePowerModes.Droop;
	UgridDroop 	: InverterMode := eInverterModes.microgrid; PowerMode :=  ePowerModes.Droop;
	UgridIsland	: InverterMode := eInverterModes.Island; PowerMode :=  ePowerModes.Droop;	
	UgridIso	: InverterMode := eInverterModes.microgrid; PowerMode :=  ePowerModes.Isochronous;	
END_CASE

//MANUAL OVERWRITES
//Overwrite for manual choice user
CASE UgridPowermode OF
	eUgridPowermode.Droop: Powermode := ePowermodes.Droop;
	eUgridPowermode.DroopZeroStart: Powermode := ePowermodes.DroopZeroStart;
	eUgridPowermode.Isochronous: Powermode := ePowermodes.Isochronous;	
END_CASE

//Overwrite for parallel setup
IF (eModeLocal = UgridIsland AND b_parallelUgrid) THEN
	InverterMode := eInvertermodes.Microgrid;
END_IF
END_METHOD

ACTION SFCTipReset:
SFCTip:= FALSE;
SFCtransTrigger.in := FALSE;
b_SFCmodetransInhibit := FALSE;
SFCResetTrigger := FALSE;
END_ACTION

METHOD ShowModeTransButton : BOOL
VAR_INPUT
END_VAR

VAR_INST
	b_ConditionalShow : BOOL;
END_VAR
CASE breakeroperationMode OF
	eBreakerOperationmode.GridFeedthrough: b_ConditionalShow := inputcontactor.b_fb;
	eBreakerOperationmode.Geniso: b_ConditionalShow := inputcontactor.b_fb AND b_hybridMode;
	ELSE
		b_ConditionalShow := FALSE;
END_CASE

ShowModeTransButton := get.b_ModeTransActive OR b_ConditionalShow;
END_METHOD

METHOD StartSequence : BOOL
VAR_INPUT
	Mode			: eBreakerOperationMode;
	b_BreakerFb		: BOOL;
	b_ACOk			: BOOL;
	b_gridFollowingmode	: BOOL;
END_VAR
VAR_OUTPUT
	SFCReset		: BOOL;
END_VAR

VAR_INST
	SequenceOption1 :  ARRAY [0..4] OF BYTE := [1,2,3,0,0];	//Warmup/start then close contactor
	SequenceOption3 :  ARRAY [0..4] OF BYTE := [2,3,0,0,0]; //Close without warmup time 
	
	ExecIndex 			: BYTE;
	b_ExtContactor		: BOOL;
	by_SequenceIndexes 	: ARRAY [0..4] OF BYTE;
	ton_ResetSEQ		: TON := (PT:= T#20S);
	b_SynchroneGenset	: BOOL;	
	b_escapeCondition	: BOOL;
	by_CurrentStep		: BYTE;

	by_RetryCounter		: BYTE;
	b_trigger			: BOOL;
	b_GenOnly			: BOOL;

	ton_SeqPulse		: TON := (PT :=T#20MS);
END_VAR
b_GenOnly:= FALSE;
SFCreset := FALSE;

CASE mode OF
  	eBreakerOperationMode.GridFeedthrough, eBreakerOperationMode.ExtGrid : 
		by_SequenceIndexes := SequenceOption3; b_SynchroneGenset := FALSE; b_escapeCondition := b_breakerFB; 
  		b_GenOnly:= FALSE;
	eBreakerOperationMode.GenDroop:  
		by_SequenceIndexes := SequenceOption1; b_SynchroneGenset := FALSE; b_escapeCondition := b_breakerFB AND b_AcOK; //b_genstarter
		b_GenOnly:= TRUE;
	eBreakerOperationMode.GenIso :  
		by_SequenceIndexes := SequenceOption1; b_SynchroneGenset := FALSE; b_escapeCondition := b_breakerFB AND b_AcOK;
		b_GenOnly:= TRUE;
	eBreakerOperationMode.GenFix :  
		by_SequenceIndexes := SequenceOption3; b_SynchroneGenset := TRUE; b_escapeCondition := b_breakerFB;
		b_GenOnly:= TRUE;
END_CASE

get.b_gensetStarting := b_GenOnly;

